# B&R Automation Studio project PT_KB_V01 (part 3)

#### FB_EH_Flow.st
```iecst
FUNCTION_BLOCK FB_EH_Flow (*TODO: FB za upravljanje elektricnim grejacima*) (*$GROUP=Pedja,$CAT=User,$GROUPICON=User.png,$CATICON=User.png*)

(* ============================================================ *)
(* 1) Inicijalizacija parametara pri rising-edge signala Enable *)
(* ============================================================ *)
IF NOT EH_Internal.Prev_Enable AND EH_Input.Enable THEN
	EH_Internal.PID_Controller.PIDParameters.Gain := EH_Constant.PID_GAIN;
	EH_Internal.PID_Controller.PIDParameters.IntegrationTime := EH_Constant.PID_INTEGRATION_TIME;
	EH_Internal.PID_Controller.PIDParameters.DerivativeTime := EH_Constant.PID_DERIVATIVE_TIME;
	EH_Internal.PID_Controller.MaxOut := EH_Constant.PID_MAX_OUT;
	EH_Internal.PID_Controller.MinOut := EH_Constant.PID_MIN_OUT;
	EH_Internal.PID_Controller.Update := TRUE;
	EH_Internal.Temp_Filter.WindowLength := EH_Constant.FILTER_LENGTH;
END_IF

IF EH_Internal.PID_Controller.UpdateDone THEN
	EH_Internal.PID_Controller.Update := TRUE;
END_IF

EH_Internal.Prev_Enable := EH_Input.Enable;

(* ================================================ *)
(* 2) Edge detekcija i priprema jednokratnih reseta *)
(* ================================================ *)
EH_Internal.Trig_Enable.CLK := EH_Input.Enable;
EH_Internal.Trig_Enable();
EH_Internal.Trig_BreakerFB_Fall.CLK := EH_Input.BreakerFB;
EH_Internal.Trig_BreakerFB_Fall();

IF EH_Internal.Trig_Enable.Q THEN
	EH_Internal.PID_Init_Pending := TRUE;
	EH_Internal.Filter_Init_Pending := TRUE;
END_IF;

(* ========================== *)
(* 3) Podesavanje svih tajmera *)
(* ========================== *)
EH_Internal.Timer_No_Flow.PT := EH_Constant.NO_FLOW_TIMEOUT;
EH_Internal.Timer_Over_Temp.PT := EH_Constant.OVER_TEMP_TIMEOUT;
EH_Internal.Timer_Breaker_On.PT := EH_Constant.BREAKER_DELAY;
EH_Internal.Timer_Breaker_Off.PT := EH_Constant.BREAKER_DELAY;

(* Svaki ciklus krecemo od FALSE, zatim po uslovima ukljucujemo IN. *)
EH_Internal.Timer_No_Flow.IN := FALSE;
EH_Internal.Timer_Over_Temp.IN := FALSE;
EH_Internal.Timer_Breaker_On.IN := FALSE;
EH_Internal.Timer_Breaker_Off.IN := FALSE;

(* ========================================================= *)
(* 4) Ogranicenje broja grejaca na validan opseg 0..MAX_HEATERS *)
(* ========================================================= *)
EH_Internal.NumHeaters_Valid := EH_Param.NumHeaters;
IF EH_Internal.NumHeaters_Valid < 0 THEN
	EH_Internal.NumHeaters_Valid := 0;
ELSIF EH_Internal.NumHeaters_Valid > EH_Constant.MAX_HEATERS THEN
	EH_Internal.NumHeaters_Valid := EH_Constant.MAX_HEATERS;
END_IF;

(* -------------------------------------------------------------------------- *)
(* 5) Validacija konfiguracije                                                 *)
(* -------------------------------------------------------------------------- *)
EH_Internal.ConfigValid := TRUE;
EH_Internal.ConfigFaultText := 'CONFIG_OK';

IF (EH_Param.OutputType <> 0) AND (EH_Param.OutputType <> 1) THEN
	EH_Internal.ConfigValid := FALSE;
	EH_Internal.ConfigFaultText := 'OutputType mora biti 0 (analog) ili 1 (PWM)';
ELSIF (EH_Param.OutputType = 0) AND (EH_Param.AnalogMin > EH_Param.AnalogMax) THEN
	EH_Internal.ConfigValid := FALSE;
	EH_Internal.ConfigFaultText := 'AnalogMin ne sme biti veci od AnalogMax';
ELSIF (EH_Param.OutputType = 1) AND (EH_Internal.NumHeaters_Valid <= 0) THEN
	EH_Internal.ConfigValid := FALSE;
	EH_Internal.ConfigFaultText := 'PWM zahteva najmanje jedan grejac';
ELSIF (EH_Param.OutputType = 1) AND (EH_Param.PWM_Width <= 0.0) THEN
	EH_Internal.ConfigValid := FALSE;
	EH_Internal.ConfigFaultText := 'PWM_Width mora biti veci od 0.0';
ELSIF (EH_Param.OutputType = 1) AND (EH_Param.ScanTime <= 0.0) THEN
	EH_Internal.ConfigValid := FALSE;
	EH_Internal.ConfigFaultText := 'ScanTime mora biti veci od 0.0 za PWM';
ELSIF EH_Param.HeaterPower < 0.0 THEN
	EH_Internal.ConfigValid := FALSE;
	EH_Internal.ConfigFaultText := 'HeaterPower ne sme biti negativan';
ELSIF EH_Param.ActiveFlowMeter AND (EH_Param.FlowNominal <= 0.0) THEN
	EH_Internal.ConfigValid := FALSE;
	EH_Internal.ConfigFaultText := 'FlowNominal mora biti veci od 0.0 uz protokomer';
END_IF;

(* =============================================== *)
(* 6) Glavna logika kada je blok omogucen (Enable) *)
(* =============================================== *)
IF EH_Input.Enable THEN
	(* Provera protoka *)
	IF EH_Param.ActiveFlowSwitch THEN
		EH_Internal.Timer_No_Flow.IN := NOT EH_Input.FlowSwitch;
	ELSIF EH_Param.ActiveFlowMeter THEN
		EH_Internal.Timer_No_Flow.IN := EH_Input.FlowRate < EH_Constant.MIN_FLOW;
	ELSE
		EH_Internal.Timer_No_Flow.IN := TRUE;  (* Alarm ako nijedan nije aktivan *)
	END_IF;

	(* Provera temperature *)
	EH_Internal.Timer_Over_Temp.IN := (EH_Input.TempOut > EH_Constant.MAX_TEMP);

	(* Havarijska situacija: gubitak BreakerFB tokom rada *)
	IF EH_Internal.Breaker_On AND EH_Internal.Trig_BreakerFB_Fall.Q THEN
		EH_Internal.Fault_Latched := TRUE;
	END_IF;

	EH_Output.Alarm := (NOT EH_Internal.ConfigValid) OR
		EH_Internal.Timer_No_Flow.Q OR EH_Internal.Timer_Over_Temp.Q;
	IF EH_Internal.Fault_Latched THEN
		EH_Output.Alarm := TRUE;
	END_IF;

	(* Sekvenca glavnog prekidaca *)
	IF NOT EH_Internal.Breaker_On THEN
		EH_Output.MainBreaker := TRUE;
		EH_Internal.Timer_Breaker_On.IN := EH_Input.BreakerFB;
		IF EH_Internal.Timer_Breaker_On.Q THEN
			EH_Internal.Breaker_On := TRUE;
		END_IF;
	END_IF;

	(* Omoguci PID i filter *)
	EH_Internal.PID_Controller.Enable := TRUE;
	EH_Internal.Temp_Filter.Enable := TRUE;

	IF EH_Output.Alarm OR NOT EH_Internal.Breaker_On THEN
		(* Iskljuci sve grejace u slucaju alarma ili ako breaker nije spreman *)
		EH_Internal.Breaker_On := FALSE;
		FOR EH_Internal.i := 0 TO EH_Constant.MAX_HEATERS-1 BY 1 DO
			EH_Output.HeaterOn[EH_Internal.i] := FALSE;
		END_FOR;
		EH_Output.AnalogOut := 0;
		EH_Output.PWMOut := 0.0;
		EH_Output.PowerConsumption := 0.0;
		EH_Internal.Demand_Percent := 0.0;
		EH_Output.Status := EH_Constant.STATUS_ALARM_OR_WAIT; (* Alarm ili breaker nije spreman *)
	ELSE
		(* Filtriranje temperature *)
		EH_Internal.Temp_Filter.Update := EH_Internal.Filter_Init_Pending;
		EH_Internal.Temp_Filter.In := EH_Input.TempOut;
		EH_Internal.Temp_Filter();
		IF EH_Internal.Filter_Init_Pending THEN
			EH_Internal.Filter_Init_Pending := FALSE;
		END_IF;

		(* PID kontrola *)
		EH_Internal.PID_Controller.IntegrationPartPresetValue := 0.0;
		EH_Internal.PID_Controller.SetIntegrationPart := EH_Internal.PID_Init_Pending;
		EH_Internal.PID_Controller.SetValue := EH_Input.Setpoint;
		EH_Internal.PID_Controller.ActValue := EH_Internal.Temp_Filter.Out;
		EH_Internal.PID_Controller();
		IF EH_Internal.PID_Init_Pending THEN
			EH_Internal.PID_Init_Pending := FALSE;
		END_IF;

		EH_Internal.Demand_Percent := EH_Internal.PID_Controller.Out;

		(* Globalni clamp da zahtev uvek ostane u opsegu 0..100% *)
		IF EH_Internal.Demand_Percent > 100.0 THEN
			EH_Internal.Demand_Percent := 100.0;
		ELSIF EH_Internal.Demand_Percent < 0.0 THEN
			EH_Internal.Demand_Percent := 0.0;
		END_IF;

		(* Korekcija za protok ako je protokomer aktivan *)
		IF EH_Param.ActiveFlowMeter AND (EH_Param.FlowNominal > 0.0) THEN
			IF EH_Input.FlowRate < EH_Param.FlowNominal THEN
				EH_Internal.Demand_Percent := EH_Internal.Demand_Percent * (EH_Input.FlowRate / EH_Param.FlowNominal);
			END_IF;
			(* Ogranici na 0-100% *)
			IF EH_Internal.Demand_Percent > 100.0 THEN
				EH_Internal.Demand_Percent := 100.0;
			ELSIF EH_Internal.Demand_Percent < 0.0 THEN
				EH_Internal.Demand_Percent := 0.0;
			END_IF;
		END_IF;

		(* Izlaz u zavisnosti od tipa *)
		CASE EH_Param.OutputType OF
			0: (* Analog *)
				EH_Output.AnalogOut := REAL_TO_INT(INT_TO_REAL(EH_Param.AnalogMin) + (INT_TO_REAL(EH_Param.AnalogMax) - INT_TO_REAL(EH_Param.AnalogMin)) * (EH_Internal.Demand_Percent / 100.0));
				EH_Output.PWMOut := 0.0;
				FOR EH_Internal.i := 0 TO EH_Internal.NumHeaters_Valid-1 BY 1 DO
					EH_Output.HeaterOn[EH_Internal.i] := TRUE;
				END_FOR;
				FOR EH_Internal.i := EH_Internal.NumHeaters_Valid TO EH_Constant.MAX_HEATERS-1 BY 1 DO
					EH_Output.HeaterOn[EH_Internal.i] := FALSE;
				END_FOR;
			1: (* PWM *)
				EH_Output.AnalogOut := 0;
				IF (EH_Internal.NumHeaters_Valid > 0) AND (EH_Param.PWM_Width > 0.0) THEN
					EH_Output.PWMOut := EH_Internal.Demand_Percent / 100.0;
					EH_Internal.Phase := EH_Internal.Phase + EH_Param.ScanTime / EH_Param.PWM_Width;
					IF EH_Internal.Phase >= 1.0 THEN
						EH_Internal.Phase := EH_Internal.Phase - 1.0;
					END_IF;
					FOR EH_Internal.i := 0 TO EH_Internal.NumHeaters_Valid-1 BY 1 DO
						EH_Internal.local_phase := EH_Internal.Phase + INT_TO_REAL(EH_Internal.i) * (1.0 / INT_TO_REAL(EH_Internal.NumHeaters_Valid));
						IF EH_Internal.local_phase >= 1.0 THEN
							EH_Internal.local_phase := EH_Internal.local_phase - 1.0;
						END_IF;
						IF EH_Internal.local_phase < EH_Internal.Demand_Percent / 100.0 THEN
							EH_Output.HeaterOn[EH_Internal.i] := TRUE;
						ELSE
							EH_Output.HeaterOn[EH_Internal.i] := FALSE;
						END_IF;
					END_FOR;
				ELSE
					(* Nedvosmislen fallback: neispravna PWM konfiguracija -> svi grejaci OFF *)
					EH_Output.PWMOut := 0.0;
					FOR EH_Internal.i := 0 TO EH_Constant.MAX_HEATERS-1 BY 1 DO
						EH_Output.HeaterOn[EH_Internal.i] := FALSE;
					END_FOR;
				END_IF;
				FOR EH_Internal.i := EH_Internal.NumHeaters_Valid TO EH_Constant.MAX_HEATERS-1 BY 1 DO
					EH_Output.HeaterOn[EH_Internal.i] := FALSE;
				END_FOR;
		ELSE
			(* Nepodrzan tip izlaza: svi izlazi se gase radi bezbednosti. *)
			EH_Output.AnalogOut := 0;
			EH_Output.PWMOut := 0.0;
			FOR EH_Internal.i := 0 TO EH_Constant.MAX_HEATERS-1 BY 1 DO
				EH_Output.HeaterOn[EH_Internal.i] := FALSE;
			END_FOR;
		END_CASE;

		(* Potrosnja energije *)
		EH_Output.PowerConsumption := INT_TO_REAL(EH_Internal.NumHeaters_Valid) * EH_Param.HeaterPower * (EH_Internal.Demand_Percent / 100.0);
		EH_Output.Status := EH_Constant.STATUS_RUNNING; (* Normalan rad *)
	END_IF;
ELSE
	(* ================================= *)
	(* 6) Logika kada je blok onemogucen *)
	(* ================================= *)
	(* Onemoguci PID i filter *)
	EH_Internal.PID_Controller.Enable := FALSE;
	EH_Internal.Temp_Filter.Enable := FALSE;
	EH_Internal.PID_Controller.SetIntegrationPart := FALSE;
	EH_Internal.Temp_Filter.Update := FALSE;

	(* Iskljuci sve kada nije omoguceno *)
	EH_Internal.Breaker_On := FALSE;
	EH_Internal.Fault_Latched := FALSE;
	EH_Internal.PID_Init_Pending := FALSE;
	EH_Internal.Filter_Init_Pending := FALSE;
	FOR EH_Internal.i := 0 TO EH_Constant.MAX_HEATERS-1  BY 1 DO
		EH_Output.HeaterOn[EH_Internal.i] := FALSE;
	END_FOR;
	EH_Output.AnalogOut := 0;
	EH_Output.PWMOut := 0.0;
	EH_Output.PowerConsumption := 0.0;
	EH_Internal.Demand_Percent := 0.0;
	EH_Output.Alarm := FALSE;
	EH_Output.Status := EH_Constant.STATUS_DISABLED; (* Blok nije aktivan *)

	(* Sekvenca iskljucivanja prekidaca *)
	EH_Internal.Timer_Breaker_Off.IN := TRUE;
	IF EH_Internal.Timer_Breaker_Off.Q THEN
		EH_Output.MainBreaker := FALSE;
	ELSE
		EH_Output.MainBreaker := TRUE;
	END_IF;
END_IF;

(* ================================================= *)
(* 7) Tekstualni opisi stanja za HMI i dijagnostiku *)
(* ================================================= *)
CASE EH_Output.Status OF
	0:
		EH_Output.StatusText := 'RUNNING_NORMAL';
	1:
		IF NOT EH_Internal.ConfigValid THEN
			EH_Output.StatusText := 'ALARM_CONFIG';
		ELSIF EH_Internal.Fault_Latched THEN
			EH_Output.StatusText := 'ALARM_BREAKER_FB';
		ELSIF EH_Internal.Timer_Over_Temp.Q THEN
			EH_Output.StatusText := 'ALARM_OVER_TEMP';
		ELSIF EH_Internal.Timer_No_Flow.Q THEN
			EH_Output.StatusText := 'ALARM_NO_FLOW';
		ELSIF NOT EH_Internal.Breaker_On THEN
			EH_Output.StatusText := 'ALARM_BREAKER_WAIT';
		ELSE
			EH_Output.StatusText := 'ALARM_GENERAL';
		END_IF;
	2:
		EH_Output.StatusText := 'DISABLED';
ELSE
	EH_Output.StatusText := 'UNKNOWN_STATUS';
END_CASE;

CASE EH_Param.OutputType OF
	0: EH_Output.OutputTypeText := 'ANALOG_OUT';
	1: EH_Output.OutputTypeText := 'PWM_OUT';
ELSE
	EH_Output.OutputTypeText := 'UNKNOWN';
END_CASE;

IF EH_Output.Status = EH_Constant.STATUS_DISABLED THEN
	EH_Output.AlarmCauseText := 'DISABLED_BY_ENABLE';
ELSIF EH_Output.Status <> EH_Constant.STATUS_ALARM_OR_WAIT THEN
	EH_Output.AlarmCauseText := 'NONE';
ELSIF NOT EH_Internal.ConfigValid THEN
	EH_Output.AlarmCauseText := 'CONFIG_INVALID';
ELSIF EH_Internal.Fault_Latched THEN
	EH_Output.AlarmCauseText := 'BREAKER_FB_LOST';
ELSIF EH_Internal.Timer_Over_Temp.Q THEN
	EH_Output.AlarmCauseText := 'OVER_TEMP';
ELSIF EH_Internal.Timer_No_Flow.Q THEN
	EH_Output.AlarmCauseText := 'NO_FLOW';
ELSIF NOT EH_Internal.Breaker_On THEN
	EH_Output.AlarmCauseText := 'BREAKER_NOT_READY';
ELSIF (EH_Param.OutputType = 1) AND ((EH_Internal.NumHeaters_Valid <= 0) OR (EH_Param.PWM_Width <= 0.0)) THEN
	EH_Output.AlarmCauseText := 'PWM_CONFIG_INVALID';
ELSIF (EH_Param.OutputType <> 0) AND (EH_Param.OutputType <> 1) THEN
	EH_Output.AlarmCauseText := 'INVALID_OUTPUT_TYPE';
ELSE
	EH_Output.AlarmCauseText := 'ALARM';
END_IF;

EH_Output.ConfigValid := EH_Internal.ConfigValid;
EH_Output.ConfigFaultText := EH_Internal.ConfigFaultText;

(* Standardni izlazi State i State_comment uskladjeni sa Status logikom. *)
CASE EH_Output.Status OF
	0:
		EH_Output.State := 1;
		EH_Output.State_comment := 'ST_ACTIVE - normalan rad protocnog grejaca';
	1:
		EH_Output.State := 2;
		EH_Output.State_comment := 'ST_ALARM_OR_WAIT - cekanje uslova ili aktivan alarm';
	2:
		EH_Output.State := 0;
		EH_Output.State_comment := 'ST_DISABLED - blok nije omogucen';
ELSE
	EH_Output.State := 255;
	EH_Output.State_comment := 'ST_UNKNOWN - nepoznato stanje';
END_CASE;

(* Pozovi tajmere *)
EH_Internal.Timer_No_Flow();
EH_Internal.Timer_Over_Temp();
EH_Internal.Timer_Breaker_On();
EH_Internal.Timer_Breaker_Off();

END_FUNCTION_BLOCK
```

#### FB_HV_2LS.st
```iecst
FUNCTION_BLOCK FB_HV_2LS (* Rucni ventil sa dva krajnja prekidaca *)

(* -------------------------------------------------------------------------- *)
(* 1) Sirovi DI uslovi i validnost polozaja                                   *)
(* -------------------------------------------------------------------------- *)
Internal.BothActiveRaw := HV_Input.CloseFb AND HV_Input.OpenFb;
Internal.TransitionRaw := (NOT HV_Input.CloseFb) AND (NOT HV_Input.OpenFb);

HV_Output.Closed := HV_Input.CloseFb AND (NOT HV_Input.OpenFb);
HV_Output.Opened := HV_Input.OpenFb AND (NOT HV_Input.CloseFb);
HV_Output.Intermediate := Internal.TransitionRaw;
HV_Output.FeedbackConflict := Internal.BothActiveRaw;
HV_Output.PositionValid := HV_Output.Opened XOR HV_Output.Closed;

(* -------------------------------------------------------------------------- *)
(* 2) Validacija parametara                                                   *)
(* -------------------------------------------------------------------------- *)
Internal.ConfigValid := TRUE;
Internal.ConfigFaultText := 'CONFIG_OK';

Cfg.T_OpenClose_Valid := HV_Param.TransitionMaxTime;
Cfg.T_BothActive_Valid := HV_Param.BothActiveFilterTime;

IF HV_Param.TransitionMaxTime <= T#0ms THEN
	Internal.ConfigValid := FALSE;
	Internal.ConfigFaultText := 'TransitionMaxTime mora biti vece od T#0ms';
	Cfg.T_OpenClose_Valid := T#10s;
END_IF;

IF HV_Param.BothActiveFilterTime < T#0ms THEN
	Internal.ConfigValid := FALSE;
	IF Internal.ConfigFaultText = 'CONFIG_OK' THEN
		Internal.ConfigFaultText := 'BothActiveFilterTime ne sme biti negativan';
	END_IF;
	Cfg.T_BothActive_Valid := T#500ms;
END_IF;

(* -------------------------------------------------------------------------- *)
(* 3) Tajmeri uslova                                                           *)
(* -------------------------------------------------------------------------- *)
Internal.TonTransition.IN := HV_Input.Enable AND Internal.ConfigValid AND Internal.TransitionRaw;
Internal.TonTransition.PT := Cfg.T_OpenClose_Valid;

Internal.TonBothActive.IN := HV_Input.Enable AND Internal.ConfigValid AND Internal.BothActiveRaw;
Internal.TonBothActive.PT := Cfg.T_BothActive_Valid;

Internal.TonTransition();
Internal.TonBothActive();

(* -------------------------------------------------------------------------- *)
(* 4) Trenutni aktivni uslov (real-time)                                      *)
(* -------------------------------------------------------------------------- *)
Internal.ActiveConditionCode := Cfg.ACT_NONE;
Internal.FaultCondition := FALSE;

IF HV_Input.Enable THEN
	IF NOT Internal.ConfigValid THEN
		Internal.ActiveConditionCode := Cfg.ACT_CONFIG_INVALID;
		Internal.FaultCondition := TRUE;
	ELSIF Internal.TonBothActive.Q THEN
		Internal.ActiveConditionCode := Cfg.ACT_BOTH_ACTIVE;
		Internal.FaultCondition := TRUE;
	ELSIF Internal.TonTransition.Q THEN
		Internal.ActiveConditionCode := Cfg.ACT_TRANSITION_TIMEOUT;
		Internal.FaultCondition := TRUE;
	END_IF;
END_IF;

(* -------------------------------------------------------------------------- *)
(* 5) Latch i reset politika                                                   *)
(* -------------------------------------------------------------------------- *)
IF HV_Input.Enable AND Internal.FaultCondition THEN
	IF NOT Internal.FaultLatched THEN
		CASE Internal.ActiveConditionCode OF
			1: Internal.FaultCode := Cfg.FLT_TRANSITION_TIMEOUT;
			2: Internal.FaultCode := Cfg.FLT_BOTH_ACTIVE;
			3: Internal.FaultCode := Cfg.FLT_CONFIG_INVALID;
		ELSE
			Internal.FaultCode := Cfg.FLT_NONE;
		END_CASE;
	END_IF;
	Internal.FaultLatched := TRUE;
END_IF;

Internal.ResetAllowed := HV_Input.Enable AND Internal.ConfigValid AND
	Internal.FaultLatched AND (NOT Internal.FaultCondition) AND HV_Output.PositionValid;

IF HV_Input.ResetAlarm AND Internal.ResetAllowed THEN
	Internal.FaultLatched := FALSE;
	Internal.FaultCode := Cfg.FLT_NONE;
END_IF;

(* -------------------------------------------------------------------------- *)
(* 6) State mapiranje                                                           *)
(* -------------------------------------------------------------------------- *)
IF NOT HV_Input.Enable THEN
	Internal.Step := Cfg.ST_DISABLED;
ELSIF Internal.BothActiveRaw THEN
	(* Fizicki konflikt se prikazuje odmah; alarm je debounced preko TonBothActive. *)
	Internal.Step := Cfg.ST_FLT_BOTH_ACTIVE;
ELSIF Internal.TransitionRaw THEN
	IF Internal.TonTransition.Q THEN
		Internal.Step := Cfg.ST_FLT_TRANSITION_TIMEOUT;
	ELSE
		Internal.Step := Cfg.ST_TRANSITION;
	END_IF;
ELSIF HV_Output.Closed THEN
	Internal.Step := Cfg.ST_CLOSED;
ELSIF HV_Output.Opened THEN
	Internal.Step := Cfg.ST_OPEN;
ELSE
	Internal.Step := Cfg.ST_TRANSITION;
END_IF;

(* -------------------------------------------------------------------------- *)
(* 7) Tekstovi stanja i dijagnostike                                           *)
(* -------------------------------------------------------------------------- *)
CASE Internal.Step OF
	0: HV_Output.State_comment := 'Stanje 0: Blok neaktivan';
	1: HV_Output.State_comment := 'Stanje 1: Ventil zatvoren';
	2: HV_Output.State_comment := 'Stanje 2: Ventil otvoren';
	3: HV_Output.State_comment := 'Stanje 3: Ventil u medjupolozaju';
	4: HV_Output.State_comment := 'Stanje 4: Medjupolozaj traje predugo';
	5: HV_Output.State_comment := 'Stanje 5: Oba krajnja signala aktivna';
ELSE
	HV_Output.State_comment := 'Stanje ?: Nepoznato stanje';
END_CASE;

CASE Internal.FaultCode OF
	0: HV_Output.FaultText := 'FLT_NONE - nema memorisanog alarma';
	1: HV_Output.FaultText := 'FLT_TRANSITION_TIMEOUT - medjupolozaj predugo traje';
	2: HV_Output.FaultText := 'FLT_BOTH_ACTIVE - oba krajnja prekidaca su aktivna';
	3: HV_Output.FaultText := 'FLT_CONFIG_INVALID - nevalidna konfiguracija parametara';
ELSE
	HV_Output.FaultText := 'FLT_UNKNOWN - nepoznat memorisani kod';
END_CASE;

IF NOT HV_Input.Enable THEN
	HV_Output.Diag := 'DISABLED';
ELSIF NOT Internal.ConfigValid THEN
	HV_Output.Diag := 'CONFIG_INVALID';
ELSIF Internal.ActiveConditionCode = Cfg.ACT_BOTH_ACTIVE THEN
	HV_Output.Diag := 'BOTH_ACTIVE_ALARM';
ELSIF Internal.ActiveConditionCode = Cfg.ACT_TRANSITION_TIMEOUT THEN
	HV_Output.Diag := 'TRANSITION_TIMEOUT_ALARM';
ELSIF Internal.FaultLatched THEN
	HV_Output.Diag := 'ALARM_LATCHED_WAIT_RESET';
ELSIF Internal.BothActiveRaw THEN
	HV_Output.Diag := 'BOTH_ACTIVE_PENDING';
ELSIF Internal.TransitionRaw THEN
	HV_Output.Diag := 'TRANSITION_TIMING';
ELSIF HV_Output.Closed THEN
	HV_Output.Diag := 'READY_CLOSED';
ELSIF HV_Output.Opened THEN
	HV_Output.Diag := 'READY_OPEN';
ELSE
	HV_Output.Diag := 'STATE_UNDEFINED';
END_IF;

(* -------------------------------------------------------------------------- *)
(* 8) Izlazi                                                                    *)
(* -------------------------------------------------------------------------- *)
HV_Output.Status := HV_Input.Enable AND Internal.ConfigValid;
HV_Output.State := Internal.Step;
HV_Output.AlarmActive := Internal.FaultCondition;
HV_Output.AlarmLatched := Internal.FaultLatched;
HV_Output.FaultCode := Internal.FaultCode;
HV_Output.ActiveConditionCode := Internal.ActiveConditionCode;
HV_Output.ConfigValid := Internal.ConfigValid;
HV_Output.ConfigFaultText := Internal.ConfigFaultText;
HV_Output.ResetAllowed := Internal.ResetAllowed;

END_FUNCTION_BLOCK
```

#### FB_V_ON_OFF_FB.st
```iecst
FUNCTION_BLOCK FB_V_ON_OFF_FB (* Jednokalemni pneumatski ON/OFF ventil *)

(* -------------------------------------------------------------------------- *)
(* 1) Validacija parametara                                                   *)
(* -------------------------------------------------------------------------- *)
Cfg.OpenMinTime_Valid := V_Param.OpenMinTime;
Cfg.OpenMaxTime_Valid := V_Param.OpenMaxTime;
Cfg.CloseMinTime_Valid := V_Param.CloseMinTime;
Cfg.CloseMaxTime_Valid := V_Param.CloseMaxTime;
Cfg.StableFbDelay_Valid := V_Param.StableFbDelay;

V_Output.ConfigFaultText := 'CONFIG_OK';

IF V_Param.OpenMaxTime <= T#0ms THEN
	Cfg.OpenMaxTime_Valid := T#1s;
	V_Output.ConfigFaultText := 'OpenMaxTime mora biti veci od T#0ms';
ELSIF V_Param.CloseMaxTime <= T#0ms THEN
	Cfg.CloseMaxTime_Valid := T#1s;
	V_Output.ConfigFaultText := 'CloseMaxTime mora biti veci od T#0ms';
ELSIF V_Param.OpenMaxTime < V_Param.OpenMinTime THEN
	Cfg.OpenMaxTime_Valid := Cfg.OpenMinTime_Valid;
	V_Output.ConfigFaultText := 'OpenMaxTime mora biti veci ili jednak OpenMinTime';
ELSIF V_Param.CloseMaxTime < V_Param.CloseMinTime THEN
	Cfg.CloseMaxTime_Valid := Cfg.CloseMinTime_Valid;
	V_Output.ConfigFaultText := 'CloseMaxTime mora biti veci ili jednak CloseMinTime';
END_IF;

IF Cfg.StableFbDelay_Valid < T#0ms THEN
	Cfg.StableFbDelay_Valid := T#0ms;
	V_Output.ConfigFaultText := 'StableFbDelay ne sme biti negativan';
END_IF;

(* -------------------------------------------------------------------------- *)
(* 2) Izbor zahteva i konverzija na komandu kalema                            *)
(* -------------------------------------------------------------------------- *)
IF V_Input.EnableManual THEN
	Internal.DesiredOpen := V_Input.Open_Manual;
ELSE
	Internal.DesiredOpen := Open;
END_IF;

(* NC: energizacija otvara. NO: energizacija zatvara. *)
Internal.CmdRequest := Internal.DesiredOpen XOR V_Param.DeEnergizedOpen;

(* -------------------------------------------------------------------------- *)
(* 3) Fizicke potvrde i memorija pretpostavljenog polozaja                     *)
(* -------------------------------------------------------------------------- *)
IF V_Param.FbOpenExists AND V_Param.FbCloseExists THEN
	Internal.OpenConfirm := V_Input.OpenFb AND NOT V_Input.CloseFb;
	Internal.CloseConfirm := V_Input.CloseFb AND NOT V_Input.OpenFb;
ELSIF V_Param.FbOpenExists THEN
	Internal.OpenConfirm := V_Input.OpenFb;
	Internal.CloseConfirm := FALSE;
ELSIF V_Param.FbCloseExists THEN
	Internal.OpenConfirm := FALSE;
	Internal.CloseConfirm := V_Input.CloseFb;
ELSE
	Internal.OpenConfirm := FALSE;
	Internal.CloseConfirm := FALSE;
END_IF;

IF V_Param.FbOpenExists THEN
	Internal.OpenAssumed := FALSE;
END_IF;
IF V_Param.FbCloseExists THEN
	Internal.CloseAssumed := FALSE;
END_IF;

(* -------------------------------------------------------------------------- *)
(* 4) Tajmeri tranzicije, merenja i stabilnog feedback-a                      *)
(* -------------------------------------------------------------------------- *)
Internal.OpenMinTimer.IN := Internal.Step = Cfg.ST_OPENING;
Internal.OpenMinTimer.PT := Cfg.OpenMinTime_Valid;
Internal.OpenMaxTimer.IN := Internal.Step = Cfg.ST_OPENING;
Internal.OpenMaxTimer.PT := Cfg.OpenMaxTime_Valid;
Internal.OpenMeasureTimer.IN := Internal.Step = Cfg.ST_OPENING;
Internal.OpenMeasureTimer.PT := T#24d;

Internal.CloseMinTimer.IN := Internal.Step = Cfg.ST_CLOSING;
Internal.CloseMinTimer.PT := Cfg.CloseMinTime_Valid;
Internal.CloseMaxTimer.IN := Internal.Step = Cfg.ST_CLOSING;
Internal.CloseMaxTimer.PT := Cfg.CloseMaxTime_Valid;
Internal.CloseMeasureTimer.IN := Internal.Step = Cfg.ST_CLOSING;
Internal.CloseMeasureTimer.PT := T#24d;

Internal.StableOpenedFbTimer.IN := V_Param.FbOpenExists AND
	(Internal.Step = Cfg.ST_IDLE_OPENED) AND Internal.DesiredOpen AND
	(NOT Internal.OpenConfirm);
Internal.StableOpenedFbTimer.PT := Cfg.StableFbDelay_Valid;

Internal.StableClosedFbTimer.IN := V_Param.FbCloseExists AND
	(Internal.Step = Cfg.ST_IDLE_CLOSED) AND (NOT Internal.DesiredOpen) AND
	(NOT Internal.CloseConfirm);
Internal.StableClosedFbTimer.PT := Cfg.StableFbDelay_Valid;

Internal.OpenMinTimer();
Internal.OpenMaxTimer();
Internal.OpenMeasureTimer();
Internal.CloseMinTimer();
Internal.CloseMaxTimer();
Internal.CloseMeasureTimer();
Internal.StableOpenedFbTimer();
Internal.StableClosedFbTimer();

(* -------------------------------------------------------------------------- *)
(* 5) Blokirajuci fault i neblokirajuci feedback alarm                        *)
(* -------------------------------------------------------------------------- *)
Internal.FaultCondition := FALSE;

IF V_Input.ManualAlarm THEN
	Internal.FaultCondition := TRUE;
	Internal.FaultCode := Cfg.FLT_MANUAL_ALARM;
END_IF;

IF V_Param.FbOpenExists AND V_Param.FbCloseExists AND
	V_Input.OpenFb AND V_Input.CloseFb THEN
	Internal.FaultCondition := TRUE;
	Internal.FaultCode := Cfg.FLT_FB_CONFLICT;
END_IF;

IF V_Output.ConfigFaultText <> 'CONFIG_OK' THEN
	Internal.FaultCondition := TRUE;
	Internal.FaultCode := Cfg.FLT_TIME_CONFIG_INVALID;
END_IF;

IF Internal.FaultCondition THEN
	Internal.FaultLatched := TRUE;
	IF V_Input.EnableManual THEN
		Internal.FaultInManual := TRUE;
	END_IF;
END_IF;

Internal.StableOpenedFbError := Internal.StableOpenedFbTimer.Q;
Internal.StableClosedFbError := Internal.StableClosedFbTimer.Q;
Internal.FeedbackAlarmCondition := Internal.StableOpenedFbError OR Internal.StableClosedFbError;

IF Internal.StableOpenedFbError THEN
	Internal.FeedbackAlarmLatched := TRUE;
	Internal.FeedbackAlarmCode := Cfg.FB_ALM_STABLE_OPEN_LOST;
ELSIF Internal.StableClosedFbError THEN
	Internal.FeedbackAlarmLatched := TRUE;
	Internal.FeedbackAlarmCode := Cfg.FB_ALM_STABLE_CLOSE_LOST;
END_IF;

(* -------------------------------------------------------------------------- *)
(* 6) Reset, Stop i Enable politika                                            *)
(* -------------------------------------------------------------------------- *)
IF V_Input.ResetAlarm THEN
	IF Internal.FaultLatched AND (NOT Internal.FaultCondition) THEN
		Internal.FaultLatched := FALSE;
		Internal.FaultInManual := FALSE;
		Internal.FaultCode := Cfg.FLT_NONE;
		Internal.ReEnableRequired := TRUE;
	END_IF;

	IF Internal.FeedbackAlarmLatched AND (NOT Internal.FeedbackAlarmCondition) THEN
		Internal.FeedbackAlarmLatched := FALSE;
		Internal.FeedbackAlarmCode := Cfg.FB_ALM_NONE;
	END_IF;
END_IF;

IF V_Input.Stop THEN
	Internal.ReEnableRequired := TRUE;
	Internal.Step := Cfg.ST_STOPPED;
ELSIF NOT V_Input.Enable THEN
	Internal.ReEnableRequired := FALSE;
	Internal.Step := Cfg.ST_DISABLED;
ELSIF Internal.FaultLatched THEN
	Internal.Step := Cfg.ST_FAULT;
ELSIF Internal.ReEnableRequired THEN
	Internal.Step := Cfg.ST_WAIT_REENABLE;
ELSIF (NOT Internal.PrevEnable) AND V_Input.Enable THEN
	(* Na prvom Enable-u izvrsava se aktuelni auto/manual zahtev. *)
	IF Internal.DesiredOpen AND Internal.OpenConfirm THEN
		Internal.Step := Cfg.ST_IDLE_OPENED;
	ELSIF (NOT Internal.DesiredOpen) AND Internal.CloseConfirm THEN
		Internal.Step := Cfg.ST_IDLE_CLOSED;
	ELSIF Internal.DesiredOpen THEN
		Internal.Step := Cfg.ST_OPENING;
		Internal.OpenAssumed := FALSE;
	ELSE
		Internal.Step := Cfg.ST_CLOSING;
		Internal.CloseAssumed := FALSE;
	END_IF;
END_IF;

(* -------------------------------------------------------------------------- *)
(* 7) State machine jednokalemnog ventila                                     *)
(* -------------------------------------------------------------------------- *)
CASE Internal.Step OF
	0: (* ST_DISABLED *)
		;

	10: (* ST_IDLE_CLOSED *)
		IF Internal.DesiredOpen THEN
			Internal.Step := Cfg.ST_OPENING;
			Internal.OpenAssumed := FALSE;
			Internal.CloseAssumed := FALSE;
		END_IF;

	20: (* ST_IDLE_OPENED *)
		IF NOT Internal.DesiredOpen THEN
			Internal.Step := Cfg.ST_CLOSING;
			Internal.OpenAssumed := FALSE;
			Internal.CloseAssumed := FALSE;
		END_IF;

	30: (* ST_OPENING *)
		IF NOT Internal.DesiredOpen THEN
			Internal.Step := Cfg.ST_CLOSING;
			Internal.OpenAssumed := FALSE;
			Internal.CloseAssumed := FALSE;
		ELSIF V_Param.FbOpenExists AND Internal.OpenConfirm THEN
			IF (V_Param.OpenMinTime = T#0ms) OR Internal.OpenMinTimer.Q THEN
				Internal.Step := Cfg.ST_IDLE_OPENED;
				V_Output.LastOpenTime := UDINT_TO_REAL(TIME_TO_UDINT(Internal.OpenMeasureTimer.ET)) / 1000.0;
			ELSE
				Internal.FaultCondition := TRUE;
				Internal.FaultLatched := TRUE;
				Internal.FaultCode := Cfg.FLT_OPEN_TOO_FAST;
				Internal.Step := Cfg.ST_FAULT;
			END_IF;
		ELSIF V_Param.FbOpenExists AND Internal.OpenMaxTimer.Q THEN
			Internal.FaultCondition := TRUE;
			Internal.FaultLatched := TRUE;
			Internal.FaultCode := Cfg.FLT_OPEN_TIMEOUT;
			Internal.Step := Cfg.ST_FAULT;
		ELSIF (NOT V_Param.FbOpenExists) AND Internal.OpenMaxTimer.Q THEN
			Internal.OpenAssumed := TRUE;
			Internal.CloseAssumed := FALSE;
			V_Output.LastOpenTime := 0.0;
			Internal.Step := Cfg.ST_IDLE_OPENED;
		END_IF;

		IF V_Param.FbCloseExists AND Internal.PrevCloseFb AND (NOT V_Input.CloseFb) THEN
			V_Output.LastOpenStartTime := UDINT_TO_REAL(TIME_TO_UDINT(Internal.OpenMeasureTimer.ET)) / 1000.0;
		ELSIF NOT V_Param.FbCloseExists THEN
			V_Output.LastOpenStartTime := 0.0;
		END_IF;

	40: (* ST_CLOSING *)
		IF Internal.DesiredOpen THEN
			Internal.Step := Cfg.ST_OPENING;
			Internal.OpenAssumed := FALSE;
			Internal.CloseAssumed := FALSE;
		ELSIF V_Param.FbCloseExists AND Internal.CloseConfirm THEN
			IF (V_Param.CloseMinTime = T#0ms) OR Internal.CloseMinTimer.Q THEN
				Internal.Step := Cfg.ST_IDLE_CLOSED;
				V_Output.LastCloseTime := UDINT_TO_REAL(TIME_TO_UDINT(Internal.CloseMeasureTimer.ET)) / 1000.0;
			ELSE
				Internal.FaultCondition := TRUE;
				Internal.FaultLatched := TRUE;
				Internal.FaultCode := Cfg.FLT_CLOSE_TOO_FAST;
				Internal.Step := Cfg.ST_FAULT;
			END_IF;
		ELSIF V_Param.FbCloseExists AND Internal.CloseMaxTimer.Q THEN
			Internal.FaultCondition := TRUE;
			Internal.FaultLatched := TRUE;
			Internal.FaultCode := Cfg.FLT_CLOSE_TIMEOUT;
			Internal.Step := Cfg.ST_FAULT;
		ELSIF (NOT V_Param.FbCloseExists) AND Internal.CloseMaxTimer.Q THEN
			Internal.OpenAssumed := FALSE;
			Internal.CloseAssumed := TRUE;
			V_Output.LastCloseTime := 0.0;
			Internal.Step := Cfg.ST_IDLE_CLOSED;
		END_IF;

		IF V_Param.FbOpenExists AND Internal.PrevOpenFb AND (NOT V_Input.OpenFb) THEN
			V_Output.LastCloseStartTime := UDINT_TO_REAL(TIME_TO_UDINT(Internal.CloseMeasureTimer.ET)) / 1000.0;
		ELSIF NOT V_Param.FbOpenExists THEN
			V_Output.LastCloseStartTime := 0.0;
		END_IF;

	50: (* ST_STOPPED *)
		;

	60: (* ST_WAIT_REENABLE *)
		;

	90: (* ST_FAULT *)
		;

ELSE
	Internal.FaultCondition := TRUE;
	Internal.FaultLatched := TRUE;
	Internal.FaultCode := Cfg.FLT_FB_CONFLICT;
	Internal.Step := Cfg.ST_FAULT;
END_CASE;

(* -------------------------------------------------------------------------- *)
(* 8) Zavrsna bezbednosna primena komande                                     *)
(* -------------------------------------------------------------------------- *)
V_Output.Cmd := FALSE;

IF V_Input.Enable AND (NOT V_Input.Stop) AND
	(V_Output.ConfigFaultText = 'CONFIG_OK') AND (NOT Internal.ReEnableRequired) THEN
	IF Internal.FaultLatched THEN
		IF V_Input.ForceCmd THEN
			V_Output.Cmd := Internal.CmdRequest;
		END_IF;
	ELSE
		V_Output.Cmd := Internal.CmdRequest;
	END_IF;
END_IF;

(* -------------------------------------------------------------------------- *)
(* 9) State, fault i alarm tekstovi                                            *)
(* -------------------------------------------------------------------------- *)
CASE Internal.Step OF
	0: V_Output.State_comment := 'ST_DISABLED - FB nije omogucen';
	10: V_Output.State_comment := 'ST_IDLE_CLOSED - ventil je zatvoren';
	20: V_Output.State_comment := 'ST_IDLE_OPENED - ventil je otvoren';
	30: V_Output.State_comment := 'ST_OPENING - ventil ide ka otvorenom';
	40: V_Output.State_comment := 'ST_CLOSING - ventil ide ka zatvorenom';
	50: V_Output.State_comment := 'ST_STOPPED - operativni Stop je aktivan';
	60: V_Output.State_comment := 'ST_WAIT_REENABLE - potreban novi Enable ciklus';
	90: V_Output.State_comment := 'ST_FAULT - blokirajuci fault je aktivan';
ELSE
	V_Output.State_comment := 'ST_UNKNOWN - nepoznato stanje';
END_CASE;

CASE Internal.FaultCode OF
	0: Internal.FaultText := 'FLT_NONE - nema blokirajuceg fault-a';
	1: Internal.FaultText := 'FLT_MANUAL_ALARM - spoljni alarm je aktivan';
	2: Internal.FaultText := 'FLT_FB_CONFLICT - oba feedback-a su aktivna';
	3: Internal.FaultText := 'FLT_OPEN_TIMEOUT - nema OpenFb potvrde';
	4: Internal.FaultText := 'FLT_OPEN_TOO_FAST - OpenFb je stigao prerano';
	5: Internal.FaultText := 'FLT_CLOSE_TIMEOUT - nema CloseFb potvrde';
	6: Internal.FaultText := 'FLT_CLOSE_TOO_FAST - CloseFb je stigao prerano';
	9: Internal.FaultText := 'FLT_TIME_CONFIG_INVALID - nevalidni vremenski parametri';
ELSE
	Internal.FaultText := 'FLT_UNKNOWN - nepoznat uzrok fault-a';
END_CASE;

CASE Internal.FeedbackAlarmCode OF
	0: V_Output.FeedbackAlarmText := 'FB_ALM_NONE - nema feedback alarma';
	1: V_Output.FeedbackAlarmText := 'FB_ALM_STABLE_OPEN_LOST - proveriti OpenFb senzor';
	2: V_Output.FeedbackAlarmText := 'FB_ALM_STABLE_CLOSE_LOST - proveriti CloseFb senzor';
ELSE
	V_Output.FeedbackAlarmText := 'FB_ALM_UNKNOWN - nepoznat feedback alarm';
END_CASE;

IF Internal.FaultLatched THEN
	IF V_Input.ForceCmd AND (NOT V_Input.Stop) AND
		(V_Output.ConfigFaultText = 'CONFIG_OK') THEN
		V_Output.Diag := 'FAULT_FORCE_ACTIVE';
	ELSE
		V_Output.Diag := 'FAULT_BLOCKING_COMMAND';
	END_IF;
ELSIF Internal.FeedbackAlarmLatched THEN
	V_Output.Diag := 'FEEDBACK_ALARM_NONBLOCKING';
ELSIF Internal.Step = Cfg.ST_WAIT_REENABLE THEN
	V_Output.Diag := 'WAIT_REENABLE';
ELSIF Internal.Step = Cfg.ST_STOPPED THEN
	V_Output.Diag := 'STOP_ACTIVE';
ELSIF (Internal.Step = Cfg.ST_OPENING) OR (Internal.Step = Cfg.ST_CLOSING) THEN
	V_Output.Diag := 'IN_TRANSITION';
ELSE
	V_Output.Diag := 'READY';
END_IF;

(* -------------------------------------------------------------------------- *)
(* 10) Zavrsno mapiranje izlaza i memorije prethodnog ciklusa                  *)
(* -------------------------------------------------------------------------- *)
V_Output.Opened := Internal.OpenConfirm OR Internal.OpenAssumed;
V_Output.Closed := Internal.CloseConfirm OR Internal.CloseAssumed;
V_Output.OpenAssumed := Internal.OpenAssumed;
V_Output.CloseAssumed := Internal.CloseAssumed;
V_Output.PositionConfirmed := Internal.OpenConfirm OR Internal.CloseConfirm;
V_Output.PositionAssumed := Internal.OpenAssumed OR Internal.CloseAssumed;
V_Output.Status := V_Input.Enable AND (NOT V_Input.Stop) AND
	(NOT Internal.FaultLatched) AND (NOT Internal.ReEnableRequired);
V_Output.InTransition := (Internal.Step = Cfg.ST_OPENING) OR (Internal.Step = Cfg.ST_CLOSING);
V_Output.StopActive := V_Input.Stop;
V_Output.WaitingReEnable := Internal.Step = Cfg.ST_WAIT_REENABLE;
V_Output.ResetAllowed := (Internal.FaultLatched AND (NOT Internal.FaultCondition)) OR
	(Internal.FeedbackAlarmLatched AND (NOT Internal.FeedbackAlarmCondition));
V_Output.State := Internal.Step;
V_Output.FaultLatched := Internal.FaultLatched;
V_Output.FaultCondition := Internal.FaultCondition;
V_Output.FaultInManual := Internal.FaultInManual;
V_Output.FaultCode := Internal.FaultCode;
V_Output.FaultText := Internal.FaultText;
V_Output.ForceActive := Internal.FaultLatched AND V_Input.ForceCmd AND
	V_Input.Enable AND (NOT V_Input.Stop) AND
	(V_Output.ConfigFaultText = 'CONFIG_OK');
V_Output.FeedbackAlarmCondition := Internal.FeedbackAlarmCondition;
V_Output.FeedbackAlarmLatched := Internal.FeedbackAlarmLatched;
V_Output.FeedbackAlarmCode := Internal.FeedbackAlarmCode;

Opened := V_Output.Opened;
Closed := V_Output.Closed;

Internal.PrevEnable := V_Input.Enable;
Internal.PrevCloseFb := V_Input.CloseFb;
Internal.PrevOpenFb := V_Input.OpenFb;

END_FUNCTION_BLOCK
```

#### FB_V_EMV.st
```iecst
FUNCTION_BLOCK FB_V_EMV (* Elektromotorni ventil sa odvojenim OPEN/CLOSE komandama *)

(* -------------------------------------------------------------------------- *)
(* 1) Podrazumevane vrednosti i izbor aktivnog zahteva                       *)
(* -------------------------------------------------------------------------- *)
V_Output.CmdOpen := FALSE;
V_Output.CmdClose := FALSE;

IF V_Input.EnableManual THEN
	Internal.DesiredOpen := V_Input.OpenManual;
ELSE
	Internal.DesiredOpen := Open;
END_IF;

(* -------------------------------------------------------------------------- *)
(* 2) Validacija parametara                                                   *)
(* -------------------------------------------------------------------------- *)
Cfg.OpenMaxTimeValid := V_Param.OpenMaxTime;
Cfg.CloseMaxTimeValid := V_Param.CloseMaxTime;
Cfg.DeadTimeValid := V_Param.DeadTime;
Cfg.EndLimitFilterTimeValid := V_Param.EndLimitFilterTime;
Cfg.PositionFbFilterTimeValid := V_Param.PositionFbFilterTime;
Cfg.OverTorqueFilterTimeValid := V_Param.OverTorqueFilterTime;
Cfg.PositionConfirmTimeValid := V_Param.PositionConfirmTime;
Cfg.StableFbLossTimeValid := V_Param.StableFbLossTime;

Internal.ConfigValid := TRUE;
Internal.ConfigFaultText := 'CONFIG_OK - parametri su validni';

IF V_Param.OpenMaxTime <= T#0ms THEN
	Internal.ConfigValid := FALSE;
	Internal.ConfigFaultText := 'OpenMaxTime mora biti vece od T#0ms';
ELSIF V_Param.CloseMaxTime <= T#0ms THEN
	Internal.ConfigValid := FALSE;
	Internal.ConfigFaultText := 'CloseMaxTime mora biti vece od T#0ms';
ELSIF V_Param.DeadTime < T#500ms THEN
	Internal.ConfigValid := FALSE;
	Internal.ConfigFaultText := 'DeadTime mora biti najmanje T#500ms';
ELSIF V_Param.EndLimitFilterTime < T#0ms THEN
	Internal.ConfigValid := FALSE;
	Internal.ConfigFaultText := 'EndLimitFilterTime ne sme biti negativan';
ELSIF V_Param.PositionFbFilterTime < T#0ms THEN
	Internal.ConfigValid := FALSE;
	Internal.ConfigFaultText := 'PositionFbFilterTime ne sme biti negativan';
ELSIF V_Param.OverTorqueFilterTime < T#0ms THEN
	Internal.ConfigValid := FALSE;
	Internal.ConfigFaultText := 'OverTorqueFilterTime ne sme biti negativan';
ELSIF V_Param.PositionConfirmTime <= T#0ms AND
	((V_Param.LampOpenExists AND V_Param.OpenFbExists) OR
	(V_Param.LampCloseExists AND V_Param.CloseFbExists)) THEN
	Internal.ConfigValid := FALSE;
	Internal.ConfigFaultText := 'PositionConfirmTime mora biti vece od T#0ms';
ELSIF V_Param.StableFbLossTime < T#0ms THEN
	Internal.ConfigValid := FALSE;
	Internal.ConfigFaultText := 'StableFbLossTime ne sme biti negativan';
END_IF;

(* -------------------------------------------------------------------------- *)
(* 3) Filtracija fizickih ulaza                                               *)
(* -------------------------------------------------------------------------- *)
IF V_Param.LampOpenExists THEN
	Internal.LampOpenFilterTimer.IN := (V_Input.LampOpen <> Internal.LampOpenStable);
	Internal.LampOpenFilterTimer.PT := Cfg.EndLimitFilterTimeValid;
	Internal.LampOpenFilterTimer();
	IF Internal.LampOpenFilterTimer.Q THEN
		Internal.LampOpenStable := V_Input.LampOpen;
	END_IF;
ELSE
	Internal.LampOpenFilterTimer.IN := FALSE;
	Internal.LampOpenFilterTimer();
	Internal.LampOpenStable := FALSE;
END_IF;

IF V_Param.LampCloseExists THEN
	Internal.LampCloseFilterTimer.IN := (V_Input.LampClose <> Internal.LampCloseStable);
	Internal.LampCloseFilterTimer.PT := Cfg.EndLimitFilterTimeValid;
	Internal.LampCloseFilterTimer();
	IF Internal.LampCloseFilterTimer.Q THEN
		Internal.LampCloseStable := V_Input.LampClose;
	END_IF;
ELSE
	Internal.LampCloseFilterTimer.IN := FALSE;
	Internal.LampCloseFilterTimer();
	Internal.LampCloseStable := FALSE;
END_IF;

IF V_Param.OpenFbExists THEN
	Internal.OpenFbFilterTimer.IN := (V_Input.OpenFb <> Internal.OpenFbStable);
	Internal.OpenFbFilterTimer.PT := Cfg.PositionFbFilterTimeValid;
	Internal.OpenFbFilterTimer();
	IF Internal.OpenFbFilterTimer.Q THEN
		Internal.OpenFbStable := V_Input.OpenFb;
	END_IF;
ELSE
	Internal.OpenFbFilterTimer.IN := FALSE;
	Internal.OpenFbFilterTimer();
	Internal.OpenFbStable := FALSE;
END_IF;

IF V_Param.CloseFbExists THEN
	Internal.CloseFbFilterTimer.IN := (V_Input.CloseFb <> Internal.CloseFbStable);
	Internal.CloseFbFilterTimer.PT := Cfg.PositionFbFilterTimeValid;
	Internal.CloseFbFilterTimer();
	IF Internal.CloseFbFilterTimer.Q THEN
		Internal.CloseFbStable := V_Input.CloseFb;
	END_IF;
ELSE
	Internal.CloseFbFilterTimer.IN := FALSE;
	Internal.CloseFbFilterTimer();
	Internal.CloseFbStable := FALSE;
END_IF;

IF V_Param.OverTorqueExists THEN
	Internal.OverTorqueFilterTimer.IN := V_Input.OverTorque;
	Internal.OverTorqueFilterTimer.PT := Cfg.OverTorqueFilterTimeValid;
	Internal.OverTorqueFilterTimer();
	Internal.OverTorqueStable := Internal.OverTorqueFilterTimer.Q;
ELSE
	Internal.OverTorqueFilterTimer.IN := FALSE;
	Internal.OverTorqueFilterTimer();
	Internal.OverTorqueStable := FALSE;
END_IF;

(* -------------------------------------------------------------------------- *)
(* 4) Tajmeri state machine                                                   *)
(* -------------------------------------------------------------------------- *)
Internal.InitSyncTimer.IN := (Internal.Step = Cfg.ST_INIT_SYNC);
Internal.InitSyncTimer.PT := Cfg.PositionFbFilterTimeValid;

Internal.DeadTimeTimer.IN := (Internal.Step = Cfg.ST_DIRECTION_DEADTIME) OR
	(Internal.Step = Cfg.ST_FORCE_DEADTIME);
Internal.DeadTimeTimer.PT := Cfg.DeadTimeValid;

Internal.OpenTravelTimer.IN := (Internal.Step = Cfg.ST_OPENING) OR
	(Internal.Step = Cfg.ST_FORCE_OPENING);
Internal.OpenTravelTimer.PT := Cfg.OpenMaxTimeValid;

Internal.CloseTravelTimer.IN := (Internal.Step = Cfg.ST_CLOSING) OR
	(Internal.Step = Cfg.ST_FORCE_CLOSING);
Internal.CloseTravelTimer.PT := Cfg.CloseMaxTimeValid;

Internal.OpenConfirmTimer.IN := (Internal.Step = Cfg.ST_WAIT_OPEN_CONFIRM) OR
	(Internal.Step = Cfg.ST_FORCE_WAIT_OPEN_CONFIRM);
Internal.OpenConfirmTimer.PT := Cfg.PositionConfirmTimeValid;

Internal.CloseConfirmTimer.IN := (Internal.Step = Cfg.ST_WAIT_CLOSE_CONFIRM) OR
	(Internal.Step = Cfg.ST_FORCE_WAIT_CLOSE_CONFIRM);
Internal.CloseConfirmTimer.PT := Cfg.PositionConfirmTimeValid;

Internal.StableOpenLossTimer.IN := V_Param.OpenFbExists AND
	(Internal.Step = Cfg.ST_IDLE_OPENED) AND (NOT Internal.OpenFbStable);
Internal.StableOpenLossTimer.PT := Cfg.StableFbLossTimeValid;

Internal.StableCloseLossTimer.IN := V_Param.CloseFbExists AND
	(Internal.Step = Cfg.ST_IDLE_CLOSED) AND (NOT Internal.CloseFbStable);
Internal.StableCloseLossTimer.PT := Cfg.StableFbLossTimeValid;

Internal.InitSyncTimer();
Internal.DeadTimeTimer();
Internal.OpenTravelTimer();
Internal.CloseTravelTimer();
Internal.OpenConfirmTimer();
Internal.CloseConfirmTimer();
Internal.StableOpenLossTimer();
Internal.StableCloseLossTimer();

(* -------------------------------------------------------------------------- *)
(* 5) Globalni fault uslovi                                                   *)
(* -------------------------------------------------------------------------- *)
Internal.FaultCondition := FALSE;

IF NOT Internal.ConfigValid THEN
	Internal.FaultCondition := TRUE;
	IF NOT Internal.FaultLatched THEN
		Internal.FaultCode := Cfg.FLT_INVALID_CONFIG;
		Internal.FaultDirection := Cfg.DIR_NONE;
	END_IF;
ELSIF V_Input.ManualAlarm THEN
	Internal.FaultCondition := TRUE;
	IF NOT Internal.FaultLatched THEN
		Internal.FaultCode := Cfg.FLT_MANUAL_ALARM;
		IF (Internal.Step = Cfg.ST_OPENING) OR (Internal.Step = Cfg.ST_FORCE_OPENING) THEN
			Internal.FaultDirection := Cfg.DIR_OPEN;
		ELSIF (Internal.Step = Cfg.ST_CLOSING) OR (Internal.Step = Cfg.ST_FORCE_CLOSING) THEN
			Internal.FaultDirection := Cfg.DIR_CLOSE;
		ELSE
			Internal.FaultDirection := Cfg.DIR_NONE;
		END_IF;
	END_IF;
ELSIF V_Param.OpenFbExists AND V_Param.CloseFbExists AND
	Internal.OpenFbStable AND Internal.CloseFbStable THEN
	Internal.FaultCondition := TRUE;
	IF NOT Internal.FaultLatched THEN
		Internal.FaultCode := Cfg.FLT_POSITION_CONFLICT;
		Internal.FaultDirection := Cfg.DIR_NONE;
	END_IF;
ELSIF V_Param.OverTorqueExists AND Internal.OverTorqueStable AND
	((Internal.Step = Cfg.ST_OPENING) OR (Internal.Step = Cfg.ST_CLOSING) OR
	(Internal.Step = Cfg.ST_FORCE_OPENING) OR (Internal.Step = Cfg.ST_FORCE_CLOSING)) THEN
	Internal.FaultCondition := TRUE;
	IF NOT Internal.FaultLatched THEN
		Internal.FaultCode := Cfg.FLT_OVER_TORQUE;
		IF (Internal.Step = Cfg.ST_OPENING) OR (Internal.Step = Cfg.ST_FORCE_OPENING) THEN
			Internal.FaultDirection := Cfg.DIR_OPEN;
		ELSE
			Internal.FaultDirection := Cfg.DIR_CLOSE;
		END_IF;
	ELSE
		Internal.RecoveryFaultCode := Cfg.FLT_OVER_TORQUE;
		Internal.FaultInForce := TRUE;
	END_IF;
ELSIF V_Param.UnexpectedOpenLimitCheck AND V_Param.LampOpenExists AND
	Internal.LampOpenStable AND
	((Internal.Step = Cfg.ST_CLOSING) OR (Internal.Step = Cfg.ST_FORCE_CLOSING)) THEN
	Internal.FaultCondition := TRUE;
	IF NOT Internal.FaultLatched THEN
		Internal.FaultCode := Cfg.FLT_UNEXPECTED_OPEN_LIMIT;
		Internal.FaultDirection := Cfg.DIR_CLOSE;
	ELSE
		Internal.RecoveryFaultCode := Cfg.FLT_UNEXPECTED_OPEN_LIMIT;
		Internal.FaultInForce := TRUE;
	END_IF;
ELSIF V_Param.UnexpectedCloseLimitCheck AND V_Param.LampCloseExists AND
	Internal.LampCloseStable AND
	((Internal.Step = Cfg.ST_OPENING) OR (Internal.Step = Cfg.ST_FORCE_OPENING)) THEN
	Internal.FaultCondition := TRUE;
	IF NOT Internal.FaultLatched THEN
		Internal.FaultCode := Cfg.FLT_UNEXPECTED_CLOSE_LIMIT;
		Internal.FaultDirection := Cfg.DIR_OPEN;
	ELSE
		Internal.RecoveryFaultCode := Cfg.FLT_UNEXPECTED_CLOSE_LIMIT;
		Internal.FaultInForce := TRUE;
	END_IF;
ELSIF Internal.StableOpenLossTimer.Q THEN
	Internal.FaultCondition := TRUE;
	IF NOT Internal.FaultLatched THEN
		Internal.FaultCode := Cfg.FLT_OPEN_FB_LOST;
		Internal.FaultDirection := Cfg.DIR_OPEN;
	END_IF;
ELSIF Internal.StableCloseLossTimer.Q THEN
	Internal.FaultCondition := TRUE;
	IF NOT Internal.FaultLatched THEN
		Internal.FaultCode := Cfg.FLT_CLOSE_FB_LOST;
		Internal.FaultDirection := Cfg.DIR_CLOSE;
	END_IF;
END_IF;

IF Internal.FaultCondition THEN
	IF NOT Internal.FaultLatched THEN
		Internal.FaultLatched := TRUE;
		Internal.FaultInManual := V_Input.EnableManual;
	END_IF;
	Internal.Step := Cfg.ST_FAULT;
END_IF;

(* -------------------------------------------------------------------------- *)
(* 6) Reset i prioritet Enable/Stop                                           *)
(* -------------------------------------------------------------------------- *)
V_Output.ResetAllowed := Internal.FaultLatched AND
	(NOT Internal.FaultCondition) AND
	(NOT V_Input.Stop) AND
	(NOT V_Input.ManualAlarm) AND
	(NOT Internal.OverTorqueStable) AND
	Internal.ConfigValid AND
	(NOT (Internal.OpenFbStable AND Internal.CloseFbStable));

IF V_Input.ResetAlarm AND V_Output.ResetAllowed THEN
	Internal.FaultLatched := FALSE;
	Internal.FaultCode := Cfg.FLT_NONE;
	Internal.FaultDirection := Cfg.DIR_NONE;
	Internal.FaultInManual := FALSE;
	Internal.FaultInForce := FALSE;
	Internal.RecoveryFaultCode := Cfg.FLT_NONE;
	IF V_Input.Enable THEN
		Internal.Step := Cfg.ST_WAIT_REENABLE;
	ELSE
		Internal.Step := Cfg.ST_DISABLED;
	END_IF;
ELSIF NOT V_Input.Enable THEN
	Internal.Step := Cfg.ST_DISABLED;
ELSIF Internal.FaultLatched AND
	(Internal.Step <> Cfg.ST_FORCE_DEADTIME) AND
	(Internal.Step <> Cfg.ST_FORCE_OPENING) AND
	(Internal.Step <> Cfg.ST_FORCE_CLOSING) AND
	(Internal.Step <> Cfg.ST_FORCE_WAIT_OPEN_CONFIRM) AND
	(Internal.Step <> Cfg.ST_FORCE_WAIT_CLOSE_CONFIRM) THEN
	Internal.Step := Cfg.ST_FAULT;
ELSIF V_Input.Stop AND (NOT Internal.FaultLatched) THEN
	Internal.Step := Cfg.ST_STOPPED;
END_IF;

(* -------------------------------------------------------------------------- *)
(* 7) Force dozvola iz fault stanja                                           *)
(* -------------------------------------------------------------------------- *)
Internal.ForceDirection := Cfg.DIR_NONE;
IF Internal.FaultDirection = Cfg.DIR_OPEN THEN
	Internal.ForceDirection := Cfg.DIR_CLOSE;
ELSIF Internal.FaultDirection = Cfg.DIR_CLOSE THEN
	Internal.ForceDirection := Cfg.DIR_OPEN;
END_IF;

Internal.ForceRequested := V_Input.ForceCmd AND
	(NOT Internal.ForceRecoveryDone) AND
	(((Internal.ForceDirection = Cfg.DIR_OPEN) AND Internal.DesiredOpen) OR
	((Internal.ForceDirection = Cfg.DIR_CLOSE) AND (NOT Internal.DesiredOpen)));

IF NOT V_Input.ForceCmd THEN
	Internal.ForceRecoveryDone := FALSE;
END_IF;

Internal.ForceAllowed := Internal.FaultLatched AND V_Input.Enable AND
	(NOT V_Input.Stop) AND Internal.ConfigValid AND
	(NOT V_Input.ManualAlarm) AND (NOT Internal.OverTorqueStable) AND
	(NOT (Internal.OpenFbStable AND Internal.CloseFbStable)) AND
	(Internal.ForceDirection <> Cfg.DIR_NONE);

(* -------------------------------------------------------------------------- *)
(* 8) State machine                                                           *)
(* -------------------------------------------------------------------------- *)
CASE Internal.Step OF
	0: (* ST_DISABLED *)
		IF V_Input.Enable AND (NOT Internal.PrevEnable) THEN
			Internal.Step := Cfg.ST_INIT_SYNC;
		END_IF;

	5: (* ST_INIT_SYNC *)
		IF Internal.InitSyncTimer.Q THEN
			IF Internal.OpenFbStable AND (NOT Internal.CloseFbStable) THEN
				IF Internal.DesiredOpen THEN
					Internal.Step := Cfg.ST_IDLE_OPENED;
				ELSE
					Internal.NextDirection := Cfg.DIR_CLOSE;
					Internal.Step := Cfg.ST_DIRECTION_DEADTIME;
				END_IF;
			ELSIF Internal.CloseFbStable AND (NOT Internal.OpenFbStable) THEN
				IF NOT Internal.DesiredOpen THEN
					Internal.Step := Cfg.ST_IDLE_CLOSED;
				ELSE
					Internal.NextDirection := Cfg.DIR_OPEN;
					Internal.Step := Cfg.ST_DIRECTION_DEADTIME;
				END_IF;
			ELSE
				IF Internal.DesiredOpen THEN
					Internal.NextDirection := Cfg.DIR_OPEN;
				ELSE
					Internal.NextDirection := Cfg.DIR_CLOSE;
				END_IF;
				Internal.Step := Cfg.ST_DIRECTION_DEADTIME;
			END_IF;
		END_IF;

	10: (* ST_IDLE_CLOSED *)
		IF Internal.DesiredOpen THEN
			Internal.NextDirection := Cfg.DIR_OPEN;
			Internal.Step := Cfg.ST_DIRECTION_DEADTIME;
		END_IF;

	20: (* ST_IDLE_OPENED *)
		IF NOT Internal.DesiredOpen THEN
			Internal.NextDirection := Cfg.DIR_CLOSE;
			Internal.Step := Cfg.ST_DIRECTION_DEADTIME;
		END_IF;

	30: (* ST_IDLE_CLOSE_ASSUMED *)
		IF Internal.DesiredOpen THEN
			Internal.NextDirection := Cfg.DIR_OPEN;
			Internal.Step := Cfg.ST_DIRECTION_DEADTIME;
		END_IF;

	40: (* ST_IDLE_OPEN_ASSUMED *)
		IF NOT Internal.DesiredOpen THEN
			Internal.NextDirection := Cfg.DIR_CLOSE;
			Internal.Step := Cfg.ST_DIRECTION_DEADTIME;
		END_IF;

	50: (* ST_INTERMEDIATE *)
		IF Internal.DesiredOpen THEN
			Internal.NextDirection := Cfg.DIR_OPEN;
		ELSE
			Internal.NextDirection := Cfg.DIR_CLOSE;
		END_IF;
		Internal.Step := Cfg.ST_DIRECTION_DEADTIME;

	60: (* ST_DIRECTION_DEADTIME *)
		IF Internal.DesiredOpen THEN
			Internal.NextDirection := Cfg.DIR_OPEN;
		ELSE
			Internal.NextDirection := Cfg.DIR_CLOSE;
		END_IF;

		IF (Internal.NextDirection = Cfg.DIR_OPEN) AND Internal.OpenFbStable THEN
			Internal.Step := Cfg.ST_IDLE_OPENED;
		ELSIF (Internal.NextDirection = Cfg.DIR_CLOSE) AND Internal.CloseFbStable THEN
			Internal.Step := Cfg.ST_IDLE_CLOSED;
		ELSIF Internal.DeadTimeTimer.Q THEN
			IF Internal.NextDirection = Cfg.DIR_OPEN THEN
				Internal.OpenEndReached := FALSE;
				Internal.OpenFbSeen := FALSE;
				Internal.OpenLampSeen := FALSE;
				Internal.OpenStartMeasured := FALSE;
				V_Output.OpenFbOffsetValid := FALSE;
				Internal.PrevDirection := Cfg.DIR_OPEN;
				Internal.Step := Cfg.ST_OPENING;
			ELSE
				Internal.CloseEndReached := FALSE;
				Internal.CloseFbSeen := FALSE;
				Internal.CloseLampSeen := FALSE;
				Internal.CloseStartMeasured := FALSE;
				V_Output.CloseFbOffsetValid := FALSE;
				Internal.PrevDirection := Cfg.DIR_CLOSE;
				Internal.Step := Cfg.ST_CLOSING;
			END_IF;
		END_IF;

	70: (* ST_OPENING *)
		IF NOT Internal.DesiredOpen THEN
			Internal.NextDirection := Cfg.DIR_CLOSE;
			Internal.Step := Cfg.ST_DIRECTION_DEADTIME;
		ELSE
			IF V_Param.OpenFbExists AND V_Input.OpenFb AND (NOT Internal.PrevOpenFbRaw) AND
				(NOT Internal.OpenFbSeen) THEN
				Internal.OpenFbEventTime := UDINT_TO_REAL(TIME_TO_UDINT(Internal.OpenTravelTimer.ET)) / 1000.0;
			END_IF;
			IF V_Param.LampOpenExists AND V_Input.LampOpen AND (NOT Internal.PrevLampOpenRaw) AND
				(NOT Internal.OpenLampSeen) THEN
				Internal.OpenLampEventTime := UDINT_TO_REAL(TIME_TO_UDINT(Internal.OpenTravelTimer.ET)) / 1000.0;
			END_IF;

			IF V_Param.CloseFbExists AND Internal.PrevCloseFbStable AND
				(NOT Internal.CloseFbStable) AND (NOT Internal.OpenStartMeasured) THEN
				V_Output.LastOpenStartTime := UDINT_TO_REAL(TIME_TO_UDINT(Internal.OpenTravelTimer.ET)) / 1000.0;
				Internal.OpenStartMeasured := TRUE;
			END_IF;

			IF V_Param.OpenFbExists AND Internal.OpenFbStable AND (NOT Internal.OpenFbSeen) THEN
				V_Output.LastOpenFbTime := Internal.OpenFbEventTime;
				Internal.OpenFbSeen := TRUE;
			END_IF;

			IF V_Param.LampOpenExists AND Internal.LampOpenStable THEN
				V_Output.LastOpenTime := Internal.OpenLampEventTime;
				Internal.OpenLampSeen := TRUE;
				Internal.OpenEndReached := TRUE;
				IF Internal.OpenFbSeen THEN
					V_Output.LastOpenFbOffset := Internal.OpenFbEventTime - Internal.OpenLampEventTime;
					V_Output.OpenFbOffsetValid := TRUE;
					Internal.Step := Cfg.ST_IDLE_OPENED;
				ELSIF V_Param.OpenFbExists THEN
					Internal.Step := Cfg.ST_WAIT_OPEN_CONFIRM;
				ELSE
					Internal.Step := Cfg.ST_IDLE_OPEN_ASSUMED;
				END_IF;
			ELSIF (NOT V_Param.LampOpenExists) AND V_Param.OpenFbExists AND Internal.OpenFbStable THEN
				V_Output.LastOpenTime := UDINT_TO_REAL(TIME_TO_UDINT(Internal.OpenTravelTimer.ET)) / 1000.0;
				Internal.Step := Cfg.ST_IDLE_OPENED;
			ELSIF Internal.OpenTravelTimer.Q THEN
				IF V_Param.LampOpenExists OR V_Param.OpenFbExists THEN
					Internal.FaultCode := Cfg.FLT_OPEN_TIMEOUT;
					Internal.FaultDirection := Cfg.DIR_OPEN;
					Internal.FaultLatched := TRUE;
					Internal.FaultInManual := V_Input.EnableManual;
					Internal.Step := Cfg.ST_FAULT;
				ELSE
					V_Output.LastOpenTime := UDINT_TO_REAL(TIME_TO_UDINT(Internal.OpenTravelTimer.ET)) / 1000.0;
					Internal.Step := Cfg.ST_IDLE_OPEN_ASSUMED;
				END_IF;
			ELSE
				V_Output.CmdOpen := TRUE;
			END_IF;
		END_IF;

	80: (* ST_CLOSING *)
		IF Internal.DesiredOpen THEN
			Internal.NextDirection := Cfg.DIR_OPEN;
			Internal.Step := Cfg.ST_DIRECTION_DEADTIME;
		ELSE
			IF V_Param.CloseFbExists AND V_Input.CloseFb AND (NOT Internal.PrevCloseFbRaw) AND
				(NOT Internal.CloseFbSeen) THEN
				Internal.CloseFbEventTime := UDINT_TO_REAL(TIME_TO_UDINT(Internal.CloseTravelTimer.ET)) / 1000.0;
			END_IF;
			IF V_Param.LampCloseExists AND V_Input.LampClose AND (NOT Internal.PrevLampCloseRaw) AND
				(NOT Internal.CloseLampSeen) THEN
				Internal.CloseLampEventTime := UDINT_TO_REAL(TIME_TO_UDINT(Internal.CloseTravelTimer.ET)) / 1000.0;
			END_IF;

			IF V_Param.OpenFbExists AND Internal.PrevOpenFbStable AND
				(NOT Internal.OpenFbStable) AND (NOT Internal.CloseStartMeasured) THEN
				V_Output.LastCloseStartTime := UDINT_TO_REAL(TIME_TO_UDINT(Internal.CloseTravelTimer.ET)) / 1000.0;
				Internal.CloseStartMeasured := TRUE;
			END_IF;

			IF V_Param.CloseFbExists AND Internal.CloseFbStable AND (NOT Internal.CloseFbSeen) THEN
				V_Output.LastCloseFbTime := Internal.CloseFbEventTime;
				Internal.CloseFbSeen := TRUE;
			END_IF;

			IF V_Param.LampCloseExists AND Internal.LampCloseStable THEN
				V_Output.LastCloseTime := Internal.CloseLampEventTime;
				Internal.CloseLampSeen := TRUE;
				Internal.CloseEndReached := TRUE;
				IF Internal.CloseFbSeen THEN
					V_Output.LastCloseFbOffset := Internal.CloseFbEventTime - Internal.CloseLampEventTime;
					V_Output.CloseFbOffsetValid := TRUE;
					Internal.Step := Cfg.ST_IDLE_CLOSED;
				ELSIF V_Param.CloseFbExists THEN
					Internal.Step := Cfg.ST_WAIT_CLOSE_CONFIRM;
				ELSE
					Internal.Step := Cfg.ST_IDLE_CLOSE_ASSUMED;
				END_IF;
			ELSIF (NOT V_Param.LampCloseExists) AND V_Param.CloseFbExists AND Internal.CloseFbStable THEN
				V_Output.LastCloseTime := UDINT_TO_REAL(TIME_TO_UDINT(Internal.CloseTravelTimer.ET)) / 1000.0;
				Internal.Step := Cfg.ST_IDLE_CLOSED;
			ELSIF Internal.CloseTravelTimer.Q THEN
				IF V_Param.LampCloseExists OR V_Param.CloseFbExists THEN
					Internal.FaultCode := Cfg.FLT_CLOSE_TIMEOUT;
					Internal.FaultDirection := Cfg.DIR_CLOSE;
					Internal.FaultLatched := TRUE;
					Internal.FaultInManual := V_Input.EnableManual;
					Internal.Step := Cfg.ST_FAULT;
				ELSE
					V_Output.LastCloseTime := UDINT_TO_REAL(TIME_TO_UDINT(Internal.CloseTravelTimer.ET)) / 1000.0;
					Internal.Step := Cfg.ST_IDLE_CLOSE_ASSUMED;
				END_IF;
			ELSE
				V_Output.CmdClose := TRUE;
			END_IF;
		END_IF;

	90: (* ST_WAIT_OPEN_CONFIRM *)
		IF Internal.OpenFbStable THEN
			Internal.OpenFbEventTime := Internal.OpenLampEventTime +
				(UDINT_TO_REAL(TIME_TO_UDINT(Internal.OpenConfirmTimer.ET)) / 1000.0);
			V_Output.LastOpenFbTime := Internal.OpenFbEventTime;
			V_Output.LastOpenFbOffset := Internal.OpenFbEventTime - Internal.OpenLampEventTime;
			V_Output.OpenFbOffsetValid := TRUE;
			Internal.Step := Cfg.ST_IDLE_OPENED;
		ELSIF Internal.OpenConfirmTimer.Q THEN
			Internal.FaultCode := Cfg.FLT_OPEN_CONFIRM_TIMEOUT;
			Internal.FaultDirection := Cfg.DIR_OPEN;
			Internal.FaultLatched := TRUE;
			Internal.FaultInManual := V_Input.EnableManual;
			Internal.Step := Cfg.ST_FAULT;
		END_IF;

	100: (* ST_WAIT_CLOSE_CONFIRM *)
		IF Internal.CloseFbStable THEN
			Internal.CloseFbEventTime := Internal.CloseLampEventTime +
				(UDINT_TO_REAL(TIME_TO_UDINT(Internal.CloseConfirmTimer.ET)) / 1000.0);
			V_Output.LastCloseFbTime := Internal.CloseFbEventTime;
			V_Output.LastCloseFbOffset := Internal.CloseFbEventTime - Internal.CloseLampEventTime;
			V_Output.CloseFbOffsetValid := TRUE;
			Internal.Step := Cfg.ST_IDLE_CLOSED;
		ELSIF Internal.CloseConfirmTimer.Q THEN
			Internal.FaultCode := Cfg.FLT_CLOSE_CONFIRM_TIMEOUT;
			Internal.FaultDirection := Cfg.DIR_CLOSE;
			Internal.FaultLatched := TRUE;
			Internal.FaultInManual := V_Input.EnableManual;
			Internal.Step := Cfg.ST_FAULT;
		END_IF;

	110: (* ST_STOPPED *)
		IF NOT V_Input.Stop THEN
			IF V_Input.Enable THEN
				Internal.Step := Cfg.ST_WAIT_REENABLE;
			ELSE
				Internal.Step := Cfg.ST_DISABLED;
			END_IF;
		END_IF;

	120: (* ST_WAIT_REENABLE *)
		(* Globalni Enable=FALSE prioritet vraca FB u ST_DISABLED. *)

	200: (* ST_FAULT *)
		IF Internal.ForceAllowed AND Internal.ForceRequested THEN
			Internal.NextDirection := Internal.ForceDirection;
			Internal.Step := Cfg.ST_FORCE_DEADTIME;
		END_IF;

	210: (* ST_FORCE_DEADTIME *)
		IF (NOT Internal.ForceAllowed) OR (NOT Internal.ForceRequested) THEN
			Internal.Step := Cfg.ST_FAULT;
		ELSIF Internal.DeadTimeTimer.Q THEN
			IF Internal.ForceDirection = Cfg.DIR_OPEN THEN
				Internal.OpenEndReached := FALSE;
				Internal.OpenFbSeen := FALSE;
				Internal.OpenLampSeen := FALSE;
				Internal.OpenStartMeasured := FALSE;
				V_Output.OpenFbOffsetValid := FALSE;
				Internal.PrevDirection := Cfg.DIR_OPEN;
				Internal.Step := Cfg.ST_FORCE_OPENING;
			ELSE
				Internal.CloseEndReached := FALSE;
				Internal.CloseFbSeen := FALSE;
				Internal.CloseLampSeen := FALSE;
				Internal.CloseStartMeasured := FALSE;
				V_Output.CloseFbOffsetValid := FALSE;
				Internal.PrevDirection := Cfg.DIR_CLOSE;
				Internal.Step := Cfg.ST_FORCE_CLOSING;
			END_IF;
		END_IF;

	220: (* ST_FORCE_OPENING *)
		IF (NOT Internal.ForceAllowed) OR (NOT Internal.ForceRequested) THEN
			Internal.Step := Cfg.ST_FAULT;
		ELSE
			IF V_Param.OpenFbExists AND V_Input.OpenFb AND (NOT Internal.PrevOpenFbRaw) AND
				(NOT Internal.OpenFbSeen) THEN
				Internal.OpenFbEventTime := UDINT_TO_REAL(TIME_TO_UDINT(Internal.OpenTravelTimer.ET)) / 1000.0;
			END_IF;
			IF V_Param.LampOpenExists AND V_Input.LampOpen AND (NOT Internal.PrevLampOpenRaw) AND
				(NOT Internal.OpenLampSeen) THEN
				Internal.OpenLampEventTime := UDINT_TO_REAL(TIME_TO_UDINT(Internal.OpenTravelTimer.ET)) / 1000.0;
			END_IF;
			IF V_Param.CloseFbExists AND Internal.PrevCloseFbStable AND
				(NOT Internal.CloseFbStable) AND (NOT Internal.OpenStartMeasured) THEN
				V_Output.LastOpenStartTime := UDINT_TO_REAL(TIME_TO_UDINT(Internal.OpenTravelTimer.ET)) / 1000.0;
				Internal.OpenStartMeasured := TRUE;
			END_IF;
			IF V_Param.OpenFbExists AND Internal.OpenFbStable AND (NOT Internal.OpenFbSeen) THEN
				V_Output.LastOpenFbTime := Internal.OpenFbEventTime;
				Internal.OpenFbSeen := TRUE;
			END_IF;
			IF V_Param.LampOpenExists AND Internal.LampOpenStable THEN
				V_Output.LastOpenTime := Internal.OpenLampEventTime;
				Internal.OpenEndReached := TRUE;
				IF Internal.OpenFbSeen THEN
					V_Output.LastOpenFbOffset := Internal.OpenFbEventTime - Internal.OpenLampEventTime;
					V_Output.OpenFbOffsetValid := TRUE;
					Internal.ForceRecoveryDone := TRUE;
					Internal.Step := Cfg.ST_FAULT;
				ELSIF V_Param.OpenFbExists THEN
					Internal.Step := Cfg.ST_FORCE_WAIT_OPEN_CONFIRM;
				ELSE
					Internal.ForceRecoveryDone := TRUE;
					Internal.Step := Cfg.ST_FAULT;
				END_IF;
			ELSIF (NOT V_Param.LampOpenExists) AND V_Param.OpenFbExists AND Internal.OpenFbStable THEN
				V_Output.LastOpenTime := UDINT_TO_REAL(TIME_TO_UDINT(Internal.OpenTravelTimer.ET)) / 1000.0;
				Internal.ForceRecoveryDone := TRUE;
				Internal.Step := Cfg.ST_FAULT;
			ELSIF Internal.OpenTravelTimer.Q THEN
				IF V_Param.LampOpenExists OR V_Param.OpenFbExists THEN
					Internal.RecoveryFaultCode := Cfg.FLT_OPEN_TIMEOUT;
					Internal.FaultInForce := TRUE;
				ELSE
					Internal.ForceRecoveryDone := TRUE;
				END_IF;
				Internal.Step := Cfg.ST_FAULT;
			ELSE
				V_Output.CmdOpen := TRUE;
			END_IF;
		END_IF;

	230: (* ST_FORCE_CLOSING *)
		IF (NOT Internal.ForceAllowed) OR (NOT Internal.ForceRequested) THEN
			Internal.Step := Cfg.ST_FAULT;
		ELSE
			IF V_Param.CloseFbExists AND V_Input.CloseFb AND (NOT Internal.PrevCloseFbRaw) AND
				(NOT Internal.CloseFbSeen) THEN
				Internal.CloseFbEventTime := UDINT_TO_REAL(TIME_TO_UDINT(Internal.CloseTravelTimer.ET)) / 1000.0;
			END_IF;
			IF V_Param.LampCloseExists AND V_Input.LampClose AND (NOT Internal.PrevLampCloseRaw) AND
				(NOT Internal.CloseLampSeen) THEN
				Internal.CloseLampEventTime := UDINT_TO_REAL(TIME_TO_UDINT(Internal.CloseTravelTimer.ET)) / 1000.0;
			END_IF;
			IF V_Param.OpenFbExists AND Internal.PrevOpenFbStable AND
				(NOT Internal.OpenFbStable) AND (NOT Internal.CloseStartMeasured) THEN
				V_Output.LastCloseStartTime := UDINT_TO_REAL(TIME_TO_UDINT(Internal.CloseTravelTimer.ET)) / 1000.0;
				Internal.CloseStartMeasured := TRUE;
			END_IF;
			IF V_Param.CloseFbExists AND Internal.CloseFbStable AND (NOT Internal.CloseFbSeen) THEN
				V_Output.LastCloseFbTime := Internal.CloseFbEventTime;
				Internal.CloseFbSeen := TRUE;
			END_IF;
			IF V_Param.LampCloseExists AND Internal.LampCloseStable THEN
				V_Output.LastCloseTime := Internal.CloseLampEventTime;
				Internal.CloseEndReached := TRUE;
				IF Internal.CloseFbSeen THEN
					V_Output.LastCloseFbOffset := Internal.CloseFbEventTime - Internal.CloseLampEventTime;
					V_Output.CloseFbOffsetValid := TRUE;
					Internal.ForceRecoveryDone := TRUE;
					Internal.Step := Cfg.ST_FAULT;
				ELSIF V_Param.CloseFbExists THEN
					Internal.Step := Cfg.ST_FORCE_WAIT_CLOSE_CONFIRM;
				ELSE
					Internal.ForceRecoveryDone := TRUE;
					Internal.Step := Cfg.ST_FAULT;
				END_IF;
			ELSIF (NOT V_Param.LampCloseExists) AND V_Param.CloseFbExists AND Internal.CloseFbStable THEN
				V_Output.LastCloseTime := UDINT_TO_REAL(TIME_TO_UDINT(Internal.CloseTravelTimer.ET)) / 1000.0;
				Internal.ForceRecoveryDone := TRUE;
				Internal.Step := Cfg.ST_FAULT;
			ELSIF Internal.CloseTravelTimer.Q THEN
				IF V_Param.LampCloseExists OR V_Param.CloseFbExists THEN
					Internal.RecoveryFaultCode := Cfg.FLT_CLOSE_TIMEOUT;
					Internal.FaultInForce := TRUE;
				ELSE
					Internal.ForceRecoveryDone := TRUE;
				END_IF;
				Internal.Step := Cfg.ST_FAULT;
			ELSE
				V_Output.CmdClose := TRUE;
			END_IF;
		END_IF;

	240: (* ST_FORCE_WAIT_OPEN_CONFIRM *)
		IF Internal.OpenFbStable THEN
			Internal.OpenFbEventTime := Internal.OpenLampEventTime +
				(UDINT_TO_REAL(TIME_TO_UDINT(Internal.OpenConfirmTimer.ET)) / 1000.0);
			V_Output.LastOpenFbTime := Internal.OpenFbEventTime;
			V_Output.LastOpenFbOffset := Internal.OpenFbEventTime - Internal.OpenLampEventTime;
			V_Output.OpenFbOffsetValid := TRUE;
			Internal.ForceRecoveryDone := TRUE;
			Internal.Step := Cfg.ST_FAULT;
		ELSIF Internal.OpenConfirmTimer.Q THEN
			Internal.RecoveryFaultCode := Cfg.FLT_OPEN_CONFIRM_TIMEOUT;
			Internal.FaultInForce := TRUE;
			Internal.Step := Cfg.ST_FAULT;
		END_IF;

	250: (* ST_FORCE_WAIT_CLOSE_CONFIRM *)
		IF Internal.CloseFbStable THEN
			Internal.CloseFbEventTime := Internal.CloseLampEventTime +
				(UDINT_TO_REAL(TIME_TO_UDINT(Internal.CloseConfirmTimer.ET)) / 1000.0);
			V_Output.LastCloseFbTime := Internal.CloseFbEventTime;
			V_Output.LastCloseFbOffset := Internal.CloseFbEventTime - Internal.CloseLampEventTime;
			V_Output.CloseFbOffsetValid := TRUE;
			Internal.ForceRecoveryDone := TRUE;
			Internal.Step := Cfg.ST_FAULT;
		ELSIF Internal.CloseConfirmTimer.Q THEN
			Internal.RecoveryFaultCode := Cfg.FLT_CLOSE_CONFIRM_TIMEOUT;
			Internal.FaultInForce := TRUE;
			Internal.Step := Cfg.ST_FAULT;
		END_IF;

ELSE
	Internal.FaultCode := Cfg.FLT_OUTPUT_CONFLICT;
	Internal.FaultDirection := Cfg.DIR_NONE;
	Internal.FaultLatched := TRUE;
	Internal.Step := Cfg.ST_FAULT;
END_CASE;

(* Defensive XOR provera nakon state machine odluke. *)
IF V_Output.CmdOpen AND V_Output.CmdClose THEN
	V_Output.CmdOpen := FALSE;
	V_Output.CmdClose := FALSE;
	IF Internal.FaultLatched THEN
		Internal.RecoveryFaultCode := Cfg.FLT_OUTPUT_CONFLICT;
		Internal.FaultInForce := TRUE;
	ELSE
		Internal.FaultCode := Cfg.FLT_OUTPUT_CONFLICT;
		Internal.FaultDirection := Cfg.DIR_NONE;
		Internal.FaultLatched := TRUE;
	END_IF;
	Internal.Step := Cfg.ST_FAULT;
END_IF;

(* -------------------------------------------------------------------------- *)
(* 9) Polozaj, status i merenja                                               *)
(* -------------------------------------------------------------------------- *)
V_Output.Opened := V_Param.OpenFbExists AND Internal.OpenFbStable AND
	(NOT Internal.CloseFbStable);
V_Output.Closed := V_Param.CloseFbExists AND Internal.CloseFbStable AND
	(NOT Internal.OpenFbStable);
V_Output.OpenAssumed := (Internal.Step = Cfg.ST_IDLE_OPEN_ASSUMED);
V_Output.CloseAssumed := (Internal.Step = Cfg.ST_IDLE_CLOSE_ASSUMED);
V_Output.PositionConfirmed := V_Output.Opened OR V_Output.Closed;
V_Output.PositionAssumed := V_Output.OpenAssumed OR V_Output.CloseAssumed;
V_Output.Intermediate := (NOT V_Output.PositionConfirmed) AND
	(NOT V_Output.PositionAssumed) AND
	(NOT (Internal.OpenFbStable AND Internal.CloseFbStable));

IF Internal.OpenFbStable AND Internal.CloseFbStable THEN
	V_Output.Position := Cfg.POS_CONFLICT;
ELSIF V_Output.Closed THEN
	V_Output.Position := Cfg.POS_CLOSED_CONFIRMED;
ELSIF V_Output.Opened THEN
	V_Output.Position := Cfg.POS_OPENED_CONFIRMED;
ELSIF V_Output.CloseAssumed THEN
	V_Output.Position := Cfg.POS_CLOSED_ASSUMED;
ELSIF V_Output.OpenAssumed THEN
	V_Output.Position := Cfg.POS_OPENED_ASSUMED;
ELSIF V_Output.Intermediate THEN
	V_Output.Position := Cfg.POS_INTERMEDIATE;
ELSE
	V_Output.Position := Cfg.POS_UNKNOWN;
END_IF;

CASE V_Output.Position OF
	0: V_Output.PositionText := 'POS_UNKNOWN - polozaj nije poznat';
	1: V_Output.PositionText := 'POS_CLOSED_CONFIRMED - zatvoren, fizicki potvrdjen';
	2: V_Output.PositionText := 'POS_OPENED_CONFIRMED - otvoren, fizicki potvrdjen';
	3: V_Output.PositionText := 'POS_INTERMEDIATE - ventil je izmedju krajnjih polozaja';
	4: V_Output.PositionText := 'POS_CLOSED_ASSUMED - zatvoren, vremenski pretpostavljen';
	5: V_Output.PositionText := 'POS_OPENED_ASSUMED - otvoren, vremenski pretpostavljen';
	6: V_Output.PositionText := 'POS_CONFLICT - OpenFb i CloseFb su istovremeno aktivni';
ELSE
	V_Output.PositionText := 'POS_INVALID - nepoznat numericki kod polozaja';
END_CASE;

V_Output.Status := V_Input.Enable AND (NOT Internal.FaultLatched);
V_Output.Ready := (Internal.Step = Cfg.ST_IDLE_CLOSED) OR
	(Internal.Step = Cfg.ST_IDLE_OPENED) OR
	(Internal.Step = Cfg.ST_IDLE_CLOSE_ASSUMED) OR
	(Internal.Step = Cfg.ST_IDLE_OPEN_ASSUMED) OR
	(Internal.Step = Cfg.ST_INTERMEDIATE);
V_Output.Opening := (Internal.Step = Cfg.ST_OPENING) OR
	(Internal.Step = Cfg.ST_FORCE_OPENING);
V_Output.Closing := (Internal.Step = Cfg.ST_CLOSING) OR
	(Internal.Step = Cfg.ST_FORCE_CLOSING);
V_Output.InTransition := V_Output.Opening OR V_Output.Closing;
V_Output.Stopped := (Internal.Step = Cfg.ST_STOPPED);
V_Output.StopActive := V_Input.Stop;
V_Output.InitActive := (Internal.Step = Cfg.ST_INIT_SYNC);
V_Output.WaitingReEnable := (Internal.Step = Cfg.ST_WAIT_REENABLE);
V_Output.DeadTimeActive := (Internal.Step = Cfg.ST_DIRECTION_DEADTIME) OR
	(Internal.Step = Cfg.ST_FORCE_DEADTIME);
V_Output.WaitingPositionConfirm := (Internal.Step = Cfg.ST_WAIT_OPEN_CONFIRM) OR
	(Internal.Step = Cfg.ST_WAIT_CLOSE_CONFIRM) OR
	(Internal.Step = Cfg.ST_FORCE_WAIT_OPEN_CONFIRM) OR
	(Internal.Step = Cfg.ST_FORCE_WAIT_CLOSE_CONFIRM);
V_Output.ManualActive := V_Input.EnableManual;
V_Output.ForceAllowed := Internal.ForceAllowed;
V_Output.ForceActive := (Internal.Step = Cfg.ST_FORCE_DEADTIME) OR
	(Internal.Step = Cfg.ST_FORCE_OPENING) OR
	(Internal.Step = Cfg.ST_FORCE_CLOSING) OR
	(Internal.Step = Cfg.ST_FORCE_WAIT_OPEN_CONFIRM) OR
	(Internal.Step = Cfg.ST_FORCE_WAIT_CLOSE_CONFIRM);
V_Output.ForceBlocked := V_Input.ForceCmd AND Internal.FaultLatched AND
	((NOT Internal.ForceAllowed) OR (NOT Internal.ForceRequested));
V_Output.DesiredOpen := Internal.DesiredOpen;
V_Output.FaultCondition := Internal.FaultCondition;
V_Output.FaultLatched := Internal.FaultLatched;
V_Output.FaultCode := Internal.FaultCode;
V_Output.FaultDirection := Internal.FaultDirection;
V_Output.FaultInManual := Internal.FaultInManual;
V_Output.FaultInForce := Internal.FaultInForce;
V_Output.ForceDirection := Internal.ForceDirection;
V_Output.RecoveryFaultCode := Internal.RecoveryFaultCode;
V_Output.ConfigFaultText := Internal.ConfigFaultText;
V_Output.OpenEndReached := Internal.OpenEndReached;
V_Output.CloseEndReached := Internal.CloseEndReached;
V_Output.OpenFbStable := Internal.OpenFbStable;
V_Output.CloseFbStable := Internal.CloseFbStable;
V_Output.OverTorqueActive := Internal.OverTorqueStable;
V_Output.State := Internal.Step;

IF V_Output.Opening THEN
	V_Output.CurrentTravelTime := UDINT_TO_REAL(TIME_TO_UDINT(Internal.OpenTravelTimer.ET)) / 1000.0;
ELSIF V_Output.Closing THEN
	V_Output.CurrentTravelTime := UDINT_TO_REAL(TIME_TO_UDINT(Internal.CloseTravelTimer.ET)) / 1000.0;
ELSE
	V_Output.CurrentTravelTime := 0.0;
END_IF;

Opened := V_Output.Opened;
Closed := V_Output.Closed;

(* -------------------------------------------------------------------------- *)
(* 10) Tekstualno mapiranje state, fault i smer kodova                       *)
(* -------------------------------------------------------------------------- *)
CASE Internal.Step OF
	0: V_Output.State_comment := 'ST_DISABLED - FB nije omogucen';
	5: V_Output.State_comment := 'ST_INIT_SYNC - proverava se pocetni polozaj';
	10: V_Output.State_comment := 'ST_IDLE_CLOSED - ventil je potvrdjeno zatvoren';
	20: V_Output.State_comment := 'ST_IDLE_OPENED - ventil je potvrdjeno otvoren';
	30: V_Output.State_comment := 'ST_IDLE_CLOSE_ASSUMED - zatvoren polozaj je pretpostavljen';
	40: V_Output.State_comment := 'ST_IDLE_OPEN_ASSUMED - otvoren polozaj je pretpostavljen';
	50: V_Output.State_comment := 'ST_INTERMEDIATE - ventil miruje u medjupolozaju';
	60: V_Output.State_comment := 'ST_DIRECTION_DEADTIME - pauza pre regularnog smera';
	70: V_Output.State_comment := 'ST_OPENING - aktivno regularno otvaranje';
	80: V_Output.State_comment := 'ST_CLOSING - aktivno regularno zatvaranje';
	90: V_Output.State_comment := 'ST_WAIT_OPEN_CONFIRM - ceka se trajni OpenFb';
	100: V_Output.State_comment := 'ST_WAIT_CLOSE_CONFIRM - ceka se trajni CloseFb';
	110: V_Output.State_comment := 'ST_STOPPED - operativni Stop je aktivan';
	120: V_Output.State_comment := 'ST_WAIT_REENABLE - potreban je novi Enable ciklus';
	200: V_Output.State_comment := 'ST_FAULT - fault je latched, regularne komande su blokirane';
	210: V_Output.State_comment := 'ST_FORCE_DEADTIME - pauza pre force oporavka';
	220: V_Output.State_comment := 'ST_FORCE_OPENING - force otvaranje iz CLOSE fault-a';
	230: V_Output.State_comment := 'ST_FORCE_CLOSING - force zatvaranje iz OPEN fault-a';
	240: V_Output.State_comment := 'ST_FORCE_WAIT_OPEN_CONFIRM - force OPEN ceka OpenFb';
	250: V_Output.State_comment := 'ST_FORCE_WAIT_CLOSE_CONFIRM - force CLOSE ceka CloseFb';
ELSE
	V_Output.State_comment := 'ST_UNKNOWN - nepoznat numericki state kod';
END_CASE;

CASE Internal.FaultCode OF
	0: V_Output.FaultText := 'FLT_NONE - nema aktivnog fault-a';
	1: V_Output.FaultText := 'FLT_MANUAL_ALARM - aktivan je spoljasnji alarm/interlock';
	2: V_Output.FaultText := 'FLT_OVER_TORQUE - aktivirana je momentna zastita';
	3: V_Output.FaultText := 'FLT_POSITION_CONFLICT - OpenFb i CloseFb su istovremeno aktivni';
	4: V_Output.FaultText := 'FLT_OUTPUT_CONFLICT - CmdOpen i CmdClose su istovremeno aktivni';
	5: V_Output.FaultText := 'FLT_OPEN_TIMEOUT - OPEN kraj nije dostignut na vreme';
	6: V_Output.FaultText := 'FLT_CLOSE_TIMEOUT - CLOSE kraj nije dostignut na vreme';
	7: V_Output.FaultText := 'FLT_OPEN_CONFIRM_TIMEOUT - LampOpen bez trajnog OpenFb';
	8: V_Output.FaultText := 'FLT_CLOSE_CONFIRM_TIMEOUT - LampClose bez trajnog CloseFb';
	9: V_Output.FaultText := 'FLT_OPEN_FB_LOST - izgubljen OpenFb u otvorenom stanju';
	10: V_Output.FaultText := 'FLT_CLOSE_FB_LOST - izgubljen CloseFb u zatvorenom stanju';
	11: V_Output.FaultText := 'FLT_INVALID_CONFIG - konfiguracija parametara nije validna';
	12: V_Output.FaultText := 'FLT_UNEXPECTED_OPEN_LIMIT - LampOpen tokom zatvaranja';
	13: V_Output.FaultText := 'FLT_UNEXPECTED_CLOSE_LIMIT - LampClose tokom otvaranja';
ELSE
	V_Output.FaultText := 'FLT_UNKNOWN - nepoznat numericki fault kod';
END_CASE;

CASE Internal.RecoveryFaultCode OF
	0: V_Output.RecoveryFaultText := 'FLT_NONE - nema fault-a tokom force oporavka';
	1: V_Output.RecoveryFaultText := 'FLT_MANUAL_ALARM - alarm tokom force oporavka';
	2: V_Output.RecoveryFaultText := 'FLT_OVER_TORQUE - momentna zastita tokom force oporavka';
	3: V_Output.RecoveryFaultText := 'FLT_POSITION_CONFLICT - konflikt polozaja tokom force oporavka';
	4: V_Output.RecoveryFaultText := 'FLT_OUTPUT_CONFLICT - konflikt izlaza tokom force oporavka';
	5: V_Output.RecoveryFaultText := 'FLT_OPEN_TIMEOUT - force otvaranje nije zavrseno na vreme';
	6: V_Output.RecoveryFaultText := 'FLT_CLOSE_TIMEOUT - force zatvaranje nije zavrseno na vreme';
	7: V_Output.RecoveryFaultText := 'FLT_OPEN_CONFIRM_TIMEOUT - force OPEN bez OpenFb potvrde';
	8: V_Output.RecoveryFaultText := 'FLT_CLOSE_CONFIRM_TIMEOUT - force CLOSE bez CloseFb potvrde';
	9: V_Output.RecoveryFaultText := 'FLT_OPEN_FB_LOST - OpenFb izgubljen tokom oporavka';
	10: V_Output.RecoveryFaultText := 'FLT_CLOSE_FB_LOST - CloseFb izgubljen tokom oporavka';
	11: V_Output.RecoveryFaultText := 'FLT_INVALID_CONFIG - konfiguracija nije validna';
	12: V_Output.RecoveryFaultText := 'FLT_UNEXPECTED_OPEN_LIMIT - neocekivan LampOpen';
	13: V_Output.RecoveryFaultText := 'FLT_UNEXPECTED_CLOSE_LIMIT - neocekivan LampClose';
ELSE
	V_Output.RecoveryFaultText := 'FLT_UNKNOWN - nepoznat recovery fault kod';
END_CASE;

CASE Internal.FaultDirection OF
	0: V_Output.FaultDirectionText := 'DIR_NONE - nema smera';
	1: V_Output.FaultDirectionText := 'DIR_OPEN - otvaranje';
	2: V_Output.FaultDirectionText := 'DIR_CLOSE - zatvaranje';
ELSE
	V_Output.FaultDirectionText := 'DIR_UNKNOWN';
END_CASE;

CASE Internal.ForceDirection OF
	0: V_Output.ForceDirectionText := 'DIR_NONE - nema smera';
	1: V_Output.ForceDirectionText := 'DIR_OPEN - otvaranje';
	2: V_Output.ForceDirectionText := 'DIR_CLOSE - zatvaranje';
ELSE
	V_Output.ForceDirectionText := 'DIR_UNKNOWN';
END_CASE;

IF V_Output.ForceActive THEN
	V_Output.ForceDiag := 'FORCE_ACTIVE - aktivan kontrolisani povratni smer';
ELSIF V_Output.ForceBlocked THEN
	V_Output.ForceDiag := 'FORCE_BLOCKED - zahtev/smer ili zastitni uslovi nisu validni';
ELSIF V_Output.ForceAllowed THEN
	V_Output.ForceDiag := 'FORCE_ALLOWED - dozvoljen je samo suprotan smer';
ELSE
	V_Output.ForceDiag := 'FORCE_NOT_AVAILABLE';
END_IF;

IF Internal.FaultLatched THEN
	V_Output.Diag := V_Output.FaultText;
ELSIF V_Output.WaitingPositionConfirm THEN
	V_Output.Diag := 'WAIT_POSITION_CONFIRM';
ELSIF V_Output.DeadTimeActive THEN
	V_Output.Diag := 'DIRECTION_DEADTIME_ACTIVE';
ELSIF V_Output.Opening THEN
	V_Output.Diag := 'OPENING_WAIT_END_SIGNAL';
ELSIF V_Output.Closing THEN
	V_Output.Diag := 'CLOSING_WAIT_END_SIGNAL';
ELSE
	V_Output.Diag := V_Output.State_comment;
END_IF;

(* -------------------------------------------------------------------------- *)
(* 11) Memorija prethodnog ciklusa                                            *)
(* -------------------------------------------------------------------------- *)
Internal.PrevEnable := V_Input.Enable;
Internal.PrevOpenFbStable := Internal.OpenFbStable;
Internal.PrevCloseFbStable := Internal.CloseFbStable;
Internal.PrevOpenFbRaw := V_Input.OpenFb;
Internal.PrevCloseFbRaw := V_Input.CloseFb;
Internal.PrevLampOpenRaw := V_Input.LampOpen;
Internal.PrevLampCloseRaw := V_Input.LampClose;

END_FUNCTION_BLOCK
```

#### FBAI01_DI01.st
```iecst
FUNCTION_BLOCK FBAI01_DI01 (* Skaliranje transmitera sa AI + statusnim DI signalom *) (*$GROUP=User,$CAT=User,$GROUPICON=User.png,$CATICON=User.png*)

(* -------------------------------------------------------------------------- *)
(* 1) Podrazumevane vrednosti po scan-u                                        *)
(* -------------------------------------------------------------------------- *)
(* Podrazumevane vrednosti po scan-u. *)
AI_Output.Status := FALSE;
AI_Internal.FaultCondition := FALSE;
AI_Internal.ActiveFaultCode := AI_Constant.FLT_NONE;
AI_Internal.ConfigValid := TRUE;
AI_Internal.ConfigFaultText := '';
AI_Output.TransmitterStatusIn := AI_Input.TransmitterStatus;
AI_Internal.ResetRequest := AI_Input.ResetAlarm;

(* -------------------------------------------------------------------------- *)
(* 2) Validacija parametara i priprema raspona                                 *)
(* -------------------------------------------------------------------------- *)
(* Validacija opsega. RawMax mora biti veci od RawMin. *)
IF AI_Param.RawMax <= AI_Param.RawMin THEN
	AI_Internal.ConfigValid := FALSE;
	AI_Internal.ConfigFaultText := 'RawMax mora biti veci od RawMin';
END_IF;

(* Validacija skaliranog opsega. ScaledMax mora biti veci od ScaledMin. *)
IF AI_Internal.ConfigValid AND (AI_Param.ScaledMax <= AI_Param.ScaledMin) THEN
	AI_Internal.ConfigValid := FALSE;
	AI_Internal.ConfigFaultText := 'ScaledMax mora biti veci od ScaledMin';
END_IF;

IF AI_Internal.ConfigValid THEN
	AI_Internal.ScaleSpanRaw := INT_TO_REAL(AI_Param.RawMax - AI_Param.RawMin);
	AI_Internal.ScaleSpanScaled := AI_Param.ScaledMax - AI_Param.ScaledMin;
ELSE
	AI_Internal.ScaleSpanRaw := 0.0;
	AI_Internal.ScaleSpanScaled := 0.0;
END_IF;

(* -------------------------------------------------------------------------- *)
(* 3) Ogranicenje manual vrednosti                                             *)
(* -------------------------------------------------------------------------- *)
(* Ogranicenje manual vrednosti na opseg. *)
AI_Internal.ManualValueLimited := AI_Input.ManualValue;
IF AI_Internal.ManualValueLimited < AI_Param.ScaledMin THEN
	AI_Internal.ManualValueLimited := AI_Param.ScaledMin;
END_IF;
IF AI_Internal.ManualValueLimited > AI_Param.ScaledMax THEN
	AI_Internal.ManualValueLimited := AI_Param.ScaledMax;
END_IF;

(* -------------------------------------------------------------------------- *)
(* 4) Fault evaluacija                                                         *)
(* -------------------------------------------------------------------------- *)
IF AI_Input.Enable THEN
	IF NOT AI_Internal.ConfigValid THEN
		AI_Internal.FaultCondition := TRUE;
		AI_Internal.ActiveFaultCode := AI_Constant.FLT_CONFIG_INVALID;
	ELSIF AI_Input.ManualAlarm THEN
		AI_Internal.FaultCondition := TRUE;
		AI_Internal.ActiveFaultCode := AI_Constant.FLT_MANUAL_ALARM;
	ELSIF (NOT AI_Input.EnableManual) AND AI_Input.UnderRange THEN
		AI_Internal.FaultCondition := TRUE;
		AI_Internal.ActiveFaultCode := AI_Constant.FLT_UNDERRANGE;
	ELSIF (NOT AI_Input.EnableManual) AND AI_Input.OverRange THEN
		AI_Internal.FaultCondition := TRUE;
		AI_Internal.ActiveFaultCode := AI_Constant.FLT_OVERRANGE;
	END_IF;
END_IF;

(* Reset je dozvoljen samo kada je latch aktivan i nema aktivnog fault uslova. *)
AI_Internal.ResetAllowed := AI_Internal.FaultLatched AND (NOT AI_Internal.FaultCondition);
IF AI_Internal.ResetRequest AND AI_Internal.ResetAllowed THEN
	AI_Internal.FaultLatched := FALSE;
	AI_Internal.FaultCode := AI_Constant.FLT_NONE;
	AI_Internal.FaultText := '';
END_IF;

(* Latch fault-a pamti prvi uzrok do validnog reset-a. *)
IF AI_Internal.FaultCondition THEN
	IF NOT AI_Internal.FaultLatched THEN
		AI_Internal.FaultCode := AI_Internal.ActiveFaultCode;
		IF AI_Internal.ActiveFaultCode = AI_Constant.FLT_MANUAL_ALARM THEN
			AI_Internal.FaultText := 'ManualAlarm aktivan';
		ELSIF AI_Internal.ActiveFaultCode = AI_Constant.FLT_UNDERRANGE THEN
			AI_Internal.FaultText := 'UnderRange signal aktivan';
		ELSIF AI_Internal.ActiveFaultCode = AI_Constant.FLT_OVERRANGE THEN
			AI_Internal.FaultText := 'OverRange signal aktivan';
		ELSIF AI_Internal.ActiveFaultCode = AI_Constant.FLT_CONFIG_INVALID THEN
			AI_Internal.FaultText := AI_Internal.ConfigFaultText;
		ELSE
			AI_Internal.FaultText := 'AI fault';
		END_IF;
	END_IF;
	AI_Internal.FaultLatched := TRUE;
END_IF;

(* -------------------------------------------------------------------------- *)
(* 5) Glavna obrada kada je blok omogucen                                      *)
(* -------------------------------------------------------------------------- *)
IF NOT AI_Input.Enable THEN
	AI_Output.ScaledValue := 0.0;
	AI_Output.State := AI_Constant.ST_DISABLED;
	AI_Output.State_comment := AI_Constant.CMT_DISABLED;
	AI_Output.Status := FALSE;
	AI_Output.UnitOfMeasureOut := AI_Param.UnitOfMeasure;
ELSE
	IF AI_Input.EnableManual THEN
		AI_Output.ScaledValue := AI_Internal.ManualValueLimited;
	ELSE
		IF AI_Internal.ConfigValid AND (AI_Internal.ScaleSpanRaw > 0.0) THEN
			AI_Output.ScaledValue :=
				AI_Param.ScaledMin +
				((INT_TO_REAL(AI_Input.RawValue - AI_Param.RawMin) / AI_Internal.ScaleSpanRaw) * AI_Internal.ScaleSpanScaled);

			(* Zavrsno ogranicenje skalirane vrednosti na parametarski opseg. *)
			IF AI_Output.ScaledValue < AI_Param.ScaledMin THEN
				AI_Output.ScaledValue := AI_Param.ScaledMin;
			END_IF;
			IF AI_Output.ScaledValue > AI_Param.ScaledMax THEN
				AI_Output.ScaledValue := AI_Param.ScaledMax;
			END_IF;
		ELSE
			AI_Output.ScaledValue := AI_Param.ScaledMin;
		END_IF;
	END_IF;

	(* ---------------------------------------------------------------------- *)
	(* 6) State i status mapiranje                                             *)
	(* ---------------------------------------------------------------------- *)
	IF AI_Internal.FaultLatched AND AI_Input.EnableManual THEN
		AI_Output.State := AI_Constant.ST_MANUAL_FAULT;
		AI_Output.State_comment := AI_Constant.CMT_MANUAL_FAULT;
		AI_Output.Status := FALSE;
	ELSIF AI_Input.EnableManual THEN
		AI_Output.State := AI_Constant.ST_MANUAL;
		AI_Output.State_comment := AI_Constant.CMT_MANUAL;
		AI_Output.Status := (NOT AI_Param.EnableStatusCheck) OR AI_Input.TransmitterStatus;
	ELSIF AI_Internal.FaultLatched THEN
		AI_Output.State := AI_Constant.ST_FAULT;
		AI_Output.State_comment := AI_Constant.CMT_FAULT;
		AI_Output.Status := FALSE;
	ELSIF AI_Param.EnableStatusCheck AND (NOT AI_Input.TransmitterStatus) THEN
		AI_Output.State := AI_Constant.ST_TRANSMITTER_STATUS_0;
		AI_Output.State_comment := AI_Constant.CMT_TRANSMITTER_STATUS_0;
		AI_Output.Status := FALSE;
	ELSIF AI_Input.RawValue < AI_Param.RawMin THEN
		AI_Output.State := AI_Constant.ST_UNDERRANGE;
		AI_Output.State_comment := AI_Constant.CMT_UNDERRANGE;
		AI_Output.Status := FALSE;
	ELSIF AI_Input.RawValue > AI_Param.RawMax THEN
		AI_Output.State := AI_Constant.ST_OVERRANGE;
		AI_Output.State_comment := AI_Constant.CMT_OVERRANGE;
		AI_Output.Status := FALSE;
	ELSE
		AI_Output.State := AI_Constant.ST_ACTIVE;
		AI_Output.State_comment := AI_Constant.CMT_ACTIVE;
		AI_Output.Status := TRUE;
	END_IF;

	AI_Output.UnitOfMeasureOut := AI_Param.UnitOfMeasure;
END_IF;

(* -------------------------------------------------------------------------- *)
(* 7) Dijagnostika i prosireni izlazi                                          *)
(* -------------------------------------------------------------------------- *)
IF NOT AI_Input.Enable THEN
	AI_Internal.Diag := 'DISABLED';
ELSIF AI_Internal.FaultLatched THEN
	IF AI_Internal.FaultCode = AI_Constant.FLT_CONFIG_INVALID THEN
		AI_Internal.Diag := 'FAULT_CONFIG_INVALID';
	ELSE
		AI_Internal.Diag := 'FAULT_LATCHED';
	END_IF;
ELSIF AI_Input.EnableManual THEN
	AI_Internal.Diag := 'MANUAL_OK';
ELSIF AI_Param.EnableStatusCheck AND (NOT AI_Input.TransmitterStatus) THEN
	AI_Internal.Diag := 'TRANSMITTER_STATUS_0';
ELSIF AI_Input.RawValue < AI_Param.RawMin THEN
	AI_Internal.Diag := 'UNDERRANGE';
ELSIF AI_Input.RawValue > AI_Param.RawMax THEN
	AI_Internal.Diag := 'OVERRANGE';
ELSE
	AI_Internal.Diag := 'ACTIVE';
END_IF;

AI_Output.FaultLatched := AI_Internal.FaultLatched;
AI_Output.FaultCondition := AI_Internal.FaultCondition;
AI_Output.ResetAllowed := AI_Internal.ResetAllowed;
AI_Output.ConfigValid := AI_Internal.ConfigValid;
AI_Output.ConfigFaultText := AI_Internal.ConfigFaultText;
AI_Output.FaultCode := AI_Internal.FaultCode;
AI_Output.FaultText := AI_Internal.FaultText;
AI_Output.Diag := AI_Internal.Diag;

END_FUNCTION_BLOCK
```
